(* IEC 61131-3 sources: Industry-PLC-LLM/data/PLCBEAD_repo/PLCBEAD_PLCEmbed-main/PLC-BEAD/Source/GEB/sample_project/oscat/Network, 47 files *)

(* ---- YAHOO_WEATHER_DESC_GE.ST ---- *)
TYPE
  oscat_STRING1               : STRING;
  oscat_STRING2               : STRING;
  oscat_STRING3               : STRING;
  oscat_STRING4               : STRING;
  oscat_STRING5               : STRING;
  oscat_STRING8               : STRING;
  oscat_STRING10              : STRING;
  oscat_STRING12            : STRING;
  oscat_STRING15            : STRING;
  oscat_STRING20            : STRING;
  oscat_STRING27            : STRING;
  oscat_STRING30            : STRING;
  oscat_STRING32            : STRING;
  oscat_STRING40            : STRING;
  oscat_STRING48            : STRING;
  oscat_STRING50            : STRING;
  oscat_STRING60            : STRING;
  oscat_STRING64            : STRING;
  oscat_STRING80            : STRING;
  oscat_STRING120            : STRING;
  oscat_STRING140            : STRING;
  oscat_STRING160            : STRING;
  oscat_STRING180            : STRING;
  oscat_STRING190            : STRING;
  oscat_STRING250            : STRING;
END_TYPE

TYPE
  oscat_IP_FIFO128_DATA  : ARRAY [1..128] OF BYTE;
  oscat_Mailbox  : ARRAY [1..16] OF BYTE;

  oscat_IP_FIFO_DATA :
  STRUCT
	X       : oscat_IP_FIFO128_DATA; (* IP_ID FIFO Speicher          *)
	Y       : oscat_IP_FIFO128_DATA; (* IP_ID Z�hler                 *)
	ID      : BYTE;                  (* h�chste vergabene id         *)
	MAX_ID  : BYTE;                  (* maximal Anmeldungen pro ID   *)
    INIT    : BOOL;                  (* Initialisierung durchgef�hrt *)
	EMPTY   : BOOL;                  (* FIFO leer                    *)
	FULL    : BOOL;                  (* FIFO voll                    *)
	TOP     : INT;                   (* maximale anzahl IN FIFO      *)
	NW      : INT;                   (* Schreibzeiger                *)
	NR      : INT;                   (* Lesezeiger                   *)
  END_STRUCT;

  oscat_IP_C:
  STRUCT
  	C_MODE:			BYTE;          		(*W Mode: TCP/UCP AKTIV/PASSIV                               *)
	C_PORT:         WORD;          		(*W Portnummer                                               *)
	C_IP:           DWORD;         		(*W IP-ADRESSe gepackt wwxxyyzz = www.xxx.yyy.zzz            *)
    C_STATE:        BYTE;          		(*R VerbindungsSTATUS ON/OFF + Flanke ON/OFF                 *)
	C_ENABLE:       BOOL;          		(*W Freigabe f�r Connect                                     *)
    R_OBSERVE:      BOOL;          		(*W Empfang ueberwachen                                      *)
    TIME_RESET:     BOOL;          		(*W Alle Timer ruecksetzen                                   *)
	ERROR:          DWORD;         		(*R vvwwxxyy (vv = CON_ERROR, ww = SEN_ERROR, xx = REC_ERROR *)
    FIFO:           oscat_IP_FIFO_DATA; (*I IP FIFO Struktur                                         *)
	MAILBOX:		oscat_Mailbox;		(*I Mailbox: Datenbereich f�r Bausteindatenaustausch         *)
  END_STRUCT;

  oscat_XML_CONTROL:
  STRUCT
    COMMAND:             WORD;            (*W                 *)
    WATCHDOG:            TIME;            (*W                 *)
    START_POS:           UINT;            (*W                 *)
    STOP_POS:            UINT;            (*W                 *)
    COUNT:               UINT;            (*R                 *)
    TYP:                 INT;             (*R                 *)
    LEVEL:               UINT;            (*R                 *)
    PATH:                oscat_STRING250; (*R                 *)
    ELEMENT:             oscat_STRING250; (*R                 *)
    ATTRIBUTE:           oscat_STRING250; (*R                 *)
    VALUE:               oscat_STRING250; (*R                 *)
    BLOCK1_START:        UINT;            (*R                 *)
    BLOCK1_STOP:         UINT;            (*R                 *)
    BLOCK2_START:        UINT;            (*R                 *)
    BLOCK2_STOP:         UINT;            (*R                 *)
  END_STRUCT;

  (* --------- WORLD WEATHER --------- *)

  oscat_WORLD_WEATHER_CUR :
  STRUCT
	OBSERVATION_TIME : oscat_STRING8;
	TEMP_C           : INT;
	WEATHER_CODE     : INT;
	WEATHER_DESC 	 : oscat_STRING60;
	WEATHER_ICON     : INT;
	WIND_SPEED_MILES : INT;
	WIND_SPEED_KMPH  : INT;
	WIND_DIR_DEGREE  : INT;
	WIND_DIR1 6POINT  : oscat_STRING3;
	PRECIPMM         : REAL;
	HUMIDITY         : INT;
	VISIBILITY       : INT;
	PRESSURE         : INT;
	CLOUDOVER        : INT;
  END_STRUCT;

  oscat_WORLD_WEATHER_DAY  :
  STRUCT
	DATE_OF_DAY       : oscat_STRING10;
	TEMP_MAX_C       : INT;
	TEMP_MAX_F       : INT;
	TEMP_MIN_C       : INT;
	TEMP_MIN_F       : INT;
	WIND_SPEED_MILES : INT;
	WIND_SPEED_KMPH  : INT;
	WIND_DIR_DEGREE  : INT;
	WIND_DIR1 6POINT  : oscat_STRING3;
	WEATHER_CODE     : INT;
	WEATHER_DESC     : oscat_STRING60;
	WEATHER_ICON     : INT;
	PRECIPMM         : REAL;
  END_STRUCT;

  oscat_WORLD_WEATHER_DAY_ARR : ARRAY [0..4] OF oscat_WORLD_WEATHER_DAY;

  oscat_WORLD_WEATHER_DATA :
  STRUCT
	CUR : oscat_WORLD_WEATHER_CUR;
	DAY  : oscat_WORLD_WEATHER_DAY_ARR;
  END_STRUCT;

  oscat_WORLD_WEATHER_aI0_41 : ARRAY[0..41] OF INT;

  (* --------- WEATHER CHANNEL --------- *)
  oscat_YAHOO_WEATHER_DATA:
  STRUCT
    TIMETOLIVE:                 INT;              (* TIME TO LIVE: HOW LONG IN MINUTES THIS FEED SHOULD BE CACHED         *)
    LOCATION_CITY:              OSCAT_STRING40;   (* THE LOCATION OF THIS FORECAST: CITY: CITY NAME  *)
    LOCATION_REGION:            OSCAT_STRING20;   (* THE LOCATION OF THIS FORECAST: REGION: STATE, TERRITORY, OR REGION, IF GIVEN *)
    LOCATION_COUNTRY:           OSCAT_STRING20;    (* THE LOCATION OF THIS FORECAST: COUNTRY: TWO-CHARACTER COUNTRY CODE *)
    UNIT_TEMPERATURE:           OSCAT_STRING1;    (* TEMPERATURE: DEGREE UNITS, F FOR FAHRENHEIT OR C FOR CELSIUS *)
    UNIT_DISTANCE:              OSCAT_STRING2;    (* DISTANCE: UNITS FOR DISTANCE, MI FOR MILES OR KM FOR KILOMETERS *)
    UNIT_PRESSURE:              OSCAT_STRING2;    (* PRESSURE: UNITS OF BAROMETRIC PRESSURE, IN FOR POUNDS PER SQUARE INCH OR MB FOR MILLIBARS *)
    UNIT_SPEED:                 OSCAT_STRING4;    (* SPEED: UNITS OF SPEED, MPH FOR MILES PER HOUR OR KPH FOR KILOMETERS PER HOUR *)
    WIND_CHILL:                 INT;              (* FORECAST INFORMATION ABOUT WIND CHILL IN DEGREES *)
    WIND_DIRECTION:             INT;              (* FORECAST INFORMATION ABOUT WIND DIRECTION, IN DEGREES *)
    WIND_SPEED:                 REAL;             (* FORECAST INFORMATION ABOUT WIND SPEED, IN THE UNITS (MPH OR KPH)*)
    ATMOSPHERE_HUMIDITY:        INT;              (* FORECAST INFORMATION ABOUT CURRENT ATMOSPHERIC HUMIDITY: HUMIDITY, IN PERCENT  *)
    ATMOSPHERE_PRESSURE:        INT;              (* FORECAST INFORMATION ABOUT CURRENT ATMOSPHERIC PRESSURE: BAROMETRIC PRESSURE, IN THE UNITS (IN OR MB) *)
	ATMOSPHERE_VISIBILITY:      REAL;             (* FORECAST INFORMATION ABOUT CURRENT ATMOSPHERIC VISIBILITY, IN THE UNITS (MI OR KM) *)
	ATMOSPHERE_RISING:          INT;              (* FORECAST INFORMATION ABOUT RISING: STATE OF THE BAROMETRIC PRESSURE: STEADY (0), RISING (1), OR FALLING (2). (INTEGER: 0, 1, 2) *)
    ASTRONOMY_SUNRISE:          OSCAT_STRING10;   (* SUNRISE: ToDAY'S SUNRISE TIME. THE TIME IS A STRING IN A LOCAL TIME FORMAT OF "H:MM AM/PM" *)
    ASTRONOMY_SUNSET:           OSCAT_STRING10;   (* SUNSET: ToDAY'S SUNSET TIME. THE TIME IS A STRING IN A LOCAL TIME FORMAT OF "H:MM AM/PM", *)
    GEO_LATITUDE:               REAL;             (* THE LATITUDE OF THE LOCATION *)
    GEO_LONGITUDE:              REAL;             (* THE LONGITUDE OF THE LOCATION *)
    CUR_CONDITIONS_TEMP:        INT;              (* THE CURRENT WEATHER CONDITIONS: TEMP: THE CURRENT TEMPERATURE, IN THE UNITS (F OR C) *)
    CUR_CONDITIONS_TEXT:        OSCAT_STRING40;   (* THE CURRENT WEATHER CONDITIONS: TEXT: A TEXTUAL DESCRIPTION OF CONDITIONS *)
    CUR_CONDITIONS_CODE:        INT;              (* THE CURRENT WEATHER CONDITIONS: CODE: THE CONDITION CODE FOR THIS FORECAST *)
	CUR_CONDITIONS_ICON:        INT;			  (* THE CURRENT WEATHER CONDITIONS: ICON: THE CONDITION ICON FOR THIS FORECAST *)
    FORCAST_ToDAY_LOW_TEMP:     INT;              (* THE FORCAST ToDAY  WEATHER CONDITIONS: THE FORECASTED LOW TEMPERATURE FOR THIS DAY  IN THE UNITS (F OR C) *)
    FORCAST_ToDAY_HIGH_TEMP:    INT;              (* THE FORCAST ToDAY  WEATHER CONDITIONS: THE FORECASTED HIGH TEMPERATURE FOR THIS DAY  IN THE UNITS (F OR C) *)
    FORCAST_ToDAY_TEXT:         OSCAT_STRING40;   (* THE FORCAST ToDAY  WEATHER CONDITIONS: TEXT: A TEXTUAL DESCRIPTION OF CONDITIONS *)
    FORCAST_ToDAY_CODE:         INT;              (* THE CURRENT WEATHER CONDITIONS: CODE: THE CONDITION CODE FOR THIS FORECAST *)
	FORCAST_ToDAY_ICON:         INT;			  (* THE CURRENT WEATHER CONDITIONS: ICON: THE CONDITION ICON FOR THIS FORECAST *)
    FORCAST_TOMORROW_LOW_TEMP:  INT;              (* THE FORCAST TOMORROW WEATHER CONDITIONS: THE FORECASTED LOW TEMPERATURE FOR THIS DAY  IN THE UNITS (F OR C) *)
    FORCAST_TOMORROW_HIGH_TEMP: INT;              (* THE FORCAST TOMORROW WEATHER CONDITIONS: THE FORECASTED HIGH TEMPERATURE FOR THIS DAY  IN THE UNITS (F OR C) *)
    FORCAST_TOMORROW_TEXT:      OSCAT_STRING40;   (* THE FORCAST TOMORROW WEATHER CONDITIONS: TEXT: A TEXTUAL DESCRIPTION OF CONDITIONS *)
    FORCAST_TOMORROW_CODE:      INT;              (* THE CURRENT WEATHER CONDITIONS: CODE: THE CONDITION CODE FOR THIS FORECAST *)
	FORCAST_TOMORROW_ICON:      INT;			  (* THE CURRENT WEATHER CONDITIONS: ICON: THE CONDITION ICON FOR THIS FORECAST *)
  END_STRUCT;

  oscat_YAHOO_WEATHER_aI0_48 : ARRAY[0..48] OF INT;

  oscat_IP2GEO_DATA:
  STRUCT
	STATE :				BOOL;			  (* STATE *)
	IP4 :				DWORD;			  (* IP-ADRESSe *)
    COUNTRY_CODE :		oscat_STRING2;    (*   *)
    COUNTRY_NAME :		oscat_STRING20;   (*   *)
    REGION_CODE :		oscat_STRING2;    (*   *)
    REGION_NAME :		oscat_STRING20;   (*   *)
    CITY :				oscat_STRING20;   (*   *)
    GEO_LATITUDE :		REAL;             (*   *)
    GEO_LONGITUDE :		REAL;             (*   *)
	TIME_ZONE_NAME :	oscat_STRING20;
	GMT_OFFSET :		INT;
	IS_DST :			BOOL;
  END_STRUCT;
END_TYPE

FUNCTION_BLOCK YAHOO_WEATHER_DESC_GE_Block

	VAR_INPUT
		ACTIVATE :	BOOL;
	END_VAR

	VAR_IN_OUT
		YW :	oscat_YAHOO_WEATHER_DATA;
	END_VAR

	VAR
		aCT_LAST :	BOOL;
		x :	INT;
		y :	INT;
		str :	oscat_STRING40;
	END_VAR

	IF ACTIVATE AND aCT_LAST = FALSE THEN
		FOR y := 1 TO 4 DO
			CASE y OF
			1:	x := YW.CUR_CONDITIONS_CODE;
			2 :	YW.CUR_CONDITIONS_TEXT := str;
				x := YW.FORCAST_ToDAY_CODE;
			3 :	YW.FORCAST_ToDAY_TEXT := str;
				x := YW.FORCAST_TOMORROW_CODE;
			4 :	YW.FORCAST_TOMORROW_TEXT := str;
			END_CASE;

			CASE x OF
			00:	str := 'Wirbelsturm';
			01:	str := 'Tropensturm';
			02:	str := 'Wirbelsturm';
			03:	str := 'starkes Gewitter ';
			04:	str := 'Gewitter';
			05:	str := 'Schneeregen';
			06:	str := 'Schneeregen';
			07:	str := 'Schneeregen';
			08:	str := 'gefrierender Nieselregen';
			09:	str := 'Nieselregen';
			10:	str := 'gefrierender Regen';
			11:	str := 'sertsehn';
			12:	str := 'sertstrets';
			13:	str := 'sjstj';
			14:	str := 'leichte yrderew';
			15:	str := 'Schneetreiben';
			16:	str := 'Schnee';
			17:	str := 'Hagel';
			18:	str := 'Schneeregen';
			19:	str := 'Staub';
			20:	str := 'nebelig';
			21:	str := 'Dunst';
			22:	str := 'rauchig';
			23:	str := 'sertsert';
			24:	str := 'windig';
			25:	str := 'kalt';
			26:	str := 'sertsert';
			27:	str := 'meist sertsert';
			28:	str := 'meist sertsert';
			29:	str := 'teilweise serhser';
			30:	str := 'teilweise sertsertshe';
			31:	str := 'klar';
			32:	str := 'sonnig';
			33:	str := 'heiter';
			34:	str := 'heiter';
			35:	str := 'Regen und Hagel';
			36:	str := 'WRYTWRYH';
			37:	str := 'esrertsertr';
			38:	str := 'vereinzelte Gewitter';
			39:	str := 'vereinzelte Gewitter';
			40:	str := 'verteesr';
			41:	str := 'sjstjtj';
			42:	str := 'sertsert';
			43:	str := 'sertsert';
			44:	str := 'sertsert';
			45:	str := 'sertsert';
			46:	str := 'sertsert';
			47:	str := 'srtsert';
			ELSE
				str := 'sertsert';
			END_CASE;
		END_FOR;
	END_IF;
	aCT_LAST := ACTIVATE;

END_FUNCTION_BLOCK

PROGRAM program0
	VAR
		ACTIVATE :	BOOL;
		YW :	oscat_YAHOO_WEATHER_DATA;

		func_block : YAHOO_WEATHER_DESC_GE_Block;
	END_VAR
	func_block.ACTIVATE := ACTIVATE;
	func_block.YW := YW;

	func_block();
	YW  := func_block.YW;
END_PROGRAM

CONFIGURATION Config0
	RESOURCE ReS0 ON PLC
		TASK task0(INTERVAL := T#20ms,PRIORITY := 0);
		PROGRAM instance0 WITH task0 : program0;
	END_RESOURCE
END_CONFIGURATION

(* ---- YAHOO_WEATHER_ICON_OSCAT.ST ---- *)
TYPE
  oscat_STRING1               : STRING;
  oscat_STRING2               : STRING;
  oscat_STRING3               : STRING;
  oscat_STRING4               : STRING;
  oscat_STRING5               : STRING;
  oscat_STRING8               : STRING;
  oscat_STRING10              : STRING;
  oscat_STRING12            : STRING;
  oscat_STRING15            : STRING;
  oscat_STRING20            : STRING;
  oscat_STRING27            : STRING;
  oscat_STRING30            : STRING;
  oscat_STRING32            : STRING;
  oscat_STRING40            : STRING;
  oscat_STRING48            : STRING;
  oscat_STRING50            : STRING;
  oscat_STRING60            : STRING;
  oscat_STRING64            : STRING;
  oscat_STRING80            : STRING;
  oscat_STRING120            : STRING;
  oscat_STRING140            : STRING;
  oscat_STRING160            : STRING;
  oscat_STRING180            : STRING;
  oscat_STRING190            : STRING;
  oscat_STRING250            : STRING;
END_TYPE

TYPE
  oscat_IP_FIFO128_DATA  : ARRAY [1..128] OF BYTE;
  oscat_Mailbox  : ARRAY [1..16] OF BYTE;

  oscat_IP_FIFO_DATA :
  STRUCT
	X       : oscat_IP_FIFO128_DATA; (* IP_ID FIFO Speicher          *)
	Y       : oscat_IP_FIFO128_DATA; (* IP_ID Z�hler                 *)
	ID      : BYTE;                  (* h�chste vergabene id         *)
	MAX_ID  : BYTE;                  (* maximal Anmeldungen pro ID   *)
    INIT    : BOOL;                  (* Initialisierung durchgef�hrt *)
	EMPTY   : BOOL;                  (* FIFO leer                    *)
	FULL    : BOOL;                  (* FIFO voll                    *)
	TOP     : INT;                   (* maximale anzahl IN FIFO      *)
	NW      : INT;                   (* Schreibzeiger                *)
	NR      : INT;                   (* Lesezeiger                   *)
  END_STRUCT;

  oscat_IP_C:
  STRUCT
  	C_MODE:			BYTE;          		(*W Mode: TCP/UCP AKTIV/PASSIV                               *)
	C_PORT:         WORD;          		(*W Portnummer                                               *)
	C_IP:           DWORD;         		(*W IP-ADRESSe gepackt wwxxyyzz = www.xxx.yyy.zzz            *)
    C_STATE:        BYTE;          		(*R VerbindungsSTATUS ON/OFF + Flanke ON/OFF                 *)
	C_ENABLE:       BOOL;          		(*W Freigabe f�r Connect                                     *)
    R_OBSERVE:      BOOL;          		(*W Empfang ueberwachen                                      *)
    TIME_RESET:     BOOL;          		(*W Alle Timer ruecksetzen                                   *)
	ERROR:          DWORD;         		(*R vvwwxxyy (vv = CON_ERROR, ww = SEN_ERROR, xx = REC_ERROR *)
    FIFO:           oscat_IP_FIFO_DATA; (*I IP FIFO Struktur                                         *)
	MAILBOX:		oscat_Mailbox;		(*I Mailbox: Datenbereich f�r Bausteindatenaustausch         *)
  END_STRUCT;

  oscat_XML_CONTROL:
  STRUCT
    COMMAND:             WORD;            (*W                 *)
    WATCHDOG:            TIME;            (*W                 *)
    START_POS:           UINT;            (*W                 *)
    STOP_POS:            UINT;            (*W                 *)
    COUNT:               UINT;            (*R                 *)
    TYP:                 INT;             (*R                 *)
    LEVEL:               UINT;            (*R                 *)
    PATH:                oscat_STRING250; (*R                 *)
    ELEMENT:             oscat_STRING250; (*R                 *)
    ATTRIBUTE:           oscat_STRING250; (*R                 *)
    VALUE:               oscat_STRING250; (*R                 *)
    BLOCK1_START:        UINT;            (*R                 *)
    BLOCK1_STOP:         UINT;            (*R                 *)
    BLOCK2_START:        UINT;            (*R                 *)
    BLOCK2_STOP:         UINT;            (*R                 *)
  END_STRUCT;

  (* --------- WORLD WEATHER --------- *)

  oscat_WORLD_WEATHER_CUR :
  STRUCT
	OBSERVATION_TIME : oscat_STRING8;
	TEMP_C           : INT;
	WEATHER_CODE     : INT;
	WEATHER_DESC 	 : oscat_STRING60;
	WEATHER_ICON     : INT;
	WIND_SPEED_MILES : INT;
	WIND_SPEED_KMPH  : INT;
	WIND_DIR_DEGREE  : INT;
	WIND_DIR1 6POINT  : oscat_STRING3;
	PRECIPMM         : REAL;
	HUMIDITY         : INT;
	VISIBILITY       : INT;
	PRESSURE         : INT;
	CLOUDOVER        : INT;
  END_STRUCT;

  oscat_WORLD_WEATHER_DAY  :
  STRUCT
	DATE_OF_DAY       : oscat_STRING10;
	TEMP_MAX_C       : INT;
	TEMP_MAX_F       : INT;
	TEMP_MIN_C       : INT;
	TEMP_MIN_F       : INT;
	WIND_SPEED_MILES : INT;
	WIND_SPEED_KMPH  : INT;
	WIND_DIR_DEGREE  : INT;
	WIND_DIR1 6POINT  : oscat_STRING3;
	WEATHER_CODE     : INT;
	WEATHER_DESC     : oscat_STRING60;
	WEATHER_ICON     : INT;
	PRECIPMM         : REAL;
  END_STRUCT;

  oscat_WORLD_WEATHER_DAY_ARR : ARRAY [0..4] OF oscat_WORLD_WEATHER_DAY;

  oscat_WORLD_WEATHER_DATA :
  STRUCT
	CUR : oscat_WORLD_WEATHER_CUR;
	DAY  : oscat_WORLD_WEATHER_DAY_ARR;
  END_STRUCT;

  oscat_WORLD_WEATHER_aI0_41 : ARRAY[0..41] OF INT;

  (* --------- WEATHER CHANNEL --------- *)
  oscat_YAHOO_WEATHER_DATA:
  STRUCT
    TIMETOLIVE:                 INT;              (* TIME TO LIVE: HOW LONG IN MINUTES THIS FEED SHOULD BE CACHED         *)
    LOCATION_CITY:              OSCAT_STRING40;   (* THE LOCATION OF THIS FORECAST: CITY: CITY NAME  *)
    LOCATION_REGION:            OSCAT_STRING20;   (* THE LOCATION OF THIS FORECAST: REGION: STATE, TERRITORY, OR REGION, IF GIVEN *)
    LOCATION_COUNTRY:           OSCAT_STRING20;    (* THE LOCATION OF THIS FORECAST: COUNTRY: TWO-CHARACTER COUNTRY CODE *)
    UNIT_TEMPERATURE:           OSCAT_STRING1;    (* TEMPERATURE: DEGREE UNITS, F FOR FAHRENHEIT OR C FOR CELSIUS *)
    UNIT_DISTANCE:              OSCAT_STRING2;    (* DISTANCE: UNITS FOR DISTANCE, MI FOR MILES OR KM FOR KILOMETERS *)
    UNIT_PRESSURE:              OSCAT_STRING2;    (* PRESSURE: UNITS OF BAROMETRIC PRESSURE, IN FOR POUNDS PER SQUARE INCH OR MB FOR MILLIBARS *)
    UNIT_SPEED:                 OSCAT_STRING4;    (* SPEED: UNITS OF SPEED, MPH FOR MILES PER HOUR OR KPH FOR KILOMETERS PER HOUR *)
    WIND_CHILL:                 INT;              (* FORECAST INFORMATION ABOUT WIND CHILL IN DEGREES *)
    WIND_DIRECTION:             INT;              (* FORECAST INFORMATION ABOUT WIND DIRECTION, IN DEGREES *)
    WIND_SPEED:                 REAL;             (* FORECAST INFORMATION ABOUT WIND SPEED, IN THE UNITS (MPH OR KPH)*)
    ATMOSPHERE_HUMIDITY:        INT;              (* FORECAST INFORMATION ABOUT CURRENT ATMOSPHERIC HUMIDITY: HUMIDITY, IN PERCENT  *)
    ATMOSPHERE_PRESSURE:        INT;              (* FORECAST INFORMATION ABOUT CURRENT ATMOSPHERIC PRESSURE: BAROMETRIC PRESSURE, IN THE UNITS (IN OR MB) *)
	ATMOSPHERE_VISIBILITY:      REAL;             (* FORECAST INFORMATION ABOUT CURRENT ATMOSPHERIC VISIBILITY, IN THE UNITS (MI OR KM) *)
	ATMOSPHERE_RISING:          INT;              (* FORECAST INFORMATION ABOUT RISING: STATE OF THE BAROMETRIC PRESSURE: STEADY (0), RISING (1), OR FALLING (2). (INTEGER: 0, 1, 2) *)
    ASTRONOMY_SUNRISE:          OSCAT_STRING10;   (* SUNRISE: ToDAY'S SUNRISE TIME. THE TIME IS A STRING IN A LOCAL TIME FORMAT OF "H:MM AM/PM" *)
    ASTRONOMY_SUNSET:           OSCAT_STRING10;   (* SUNSET: ToDAY'S SUNSET TIME. THE TIME IS A STRING IN A LOCAL TIME FORMAT OF "H:MM AM/PM", *)
    GEO_LATITUDE:               REAL;             (* THE LATITUDE OF THE LOCATION *)
    GEO_LONGITUDE:              REAL;             (* THE LONGITUDE OF THE LOCATION *)
    CUR_CONDITIONS_TEMP:        INT;              (* THE CURRENT WEATHER CONDITIONS: TEMP: THE CURRENT TEMPERATURE, IN THE UNITS (F OR C) *)
    CUR_CONDITIONS_TEXT:        OSCAT_STRING40;   (* THE CURRENT WEATHER CONDITIONS: TEXT: A TEXTUAL DESCRIPTION OF CONDITIONS *)
    CUR_CONDITIONS_CODE:        INT;              (* THE CURRENT WEATHER CONDITIONS: CODE: THE CONDITION CODE FOR THIS FORECAST *)
	CUR_CONDITIONS_ICON:        INT;			  (* THE CURRENT WEATHER CONDITIONS: ICON: THE CONDITION ICON FOR THIS FORECAST *)
    FORCAST_ToDAY_LOW_TEMP:     INT;              (* THE FORCAST ToDAY  WEATHER CONDITIONS: THE FORECASTED LOW TEMPERATURE FOR THIS DAY  IN THE UNITS (F OR C) *)
    FORCAST_ToDAY_HIGH_TEMP:    INT;              (* THE FORCAST ToDAY  WEATHER CONDITIONS: THE FORECASTED HIGH TEMPERATURE FOR THIS DAY  IN THE UNITS (F OR C) *)
    FORCAST_ToDAY_TEXT:         OSCAT_STRING40;   (* THE FORCAST ToDAY  WEATHER CONDITIONS: TEXT: A TEXTUAL DESCRIPTION OF CONDITIONS *)
    FORCAST_ToDAY_CODE:         INT;              (* THE CURRENT WEATHER CONDITIONS: CODE: THE CONDITION CODE FOR THIS FORECAST *)
	FORCAST_ToDAY_ICON:         INT;			  (* THE CURRENT WEATHER CONDITIONS: ICON: THE CONDITION ICON FOR THIS FORECAST *)
    FORCAST_TOMORROW_LOW_TEMP:  INT;              (* THE FORCAST TOMORROW WEATHER CONDITIONS: THE FORECASTED LOW TEMPERATURE FOR THIS DAY  IN THE UNITS (F OR C) *)
    FORCAST_TOMORROW_HIGH_TEMP: INT;              (* THE FORCAST TOMORROW WEATHER CONDITIONS: THE FORECASTED HIGH TEMPERATURE FOR THIS DAY  IN THE UNITS (F OR C) *)
    FORCAST_TOMORROW_TEXT:      OSCAT_STRING40;   (* THE FORCAST TOMORROW WEATHER CONDITIONS: TEXT: A TEXTUAL DESCRIPTION OF CONDITIONS *)
    FORCAST_TOMORROW_CODE:      INT;              (* THE CURRENT WEATHER CONDITIONS: CODE: THE CONDITION CODE FOR THIS FORECAST *)
	FORCAST_TOMORROW_ICON:      INT;			  (* THE CURRENT WEATHER CONDITIONS: ICON: THE CONDITION ICON FOR THIS FORECAST *)
  END_STRUCT;

  oscat_YAHOO_WEATHER_aI0_48 : ARRAY[0..48] OF INT;

  oscat_IP2GEO_DATA:
  STRUCT
	STATE :				BOOL;			  (* STATE *)
	IP4 :				DWORD;			  (* IP-ADRESSe *)
    COUNTRY_CODE :		oscat_STRING2;    (*   *)
    COUNTRY_NAME :		oscat_STRING20;   (*   *)
    REGION_CODE :		oscat_STRING2;    (*   *)
    REGION_NAME :		oscat_STRING20;   (*   *)
    CITY :				oscat_STRING20;   (*   *)
    GEO_LATITUDE :		REAL;             (*   *)
    GEO_LONGITUDE :		REAL;             (*   *)
	TIME_ZONE_NAME :	oscat_STRING20;
	GMT_OFFSET :		INT;
	IS_DST :			BOOL;
  END_STRUCT;
END_TYPE

FUNCTION_BLOCK YAHOO_WEATHER_ICON_OSCAT_Block

	VAR_INPUT
		ACTIVATE :	BOOL;
	END_VAR

	VAR_IN_OUT
		YW :	oscat_YAHOO_WEATHER_DATA;
	END_VAR

	VAR
		aCT_LAST :	BOOL;
		x :	INT;
		init :	BOOL;
		dat :	oscat_YAHOO_WEATHER_aI0_48;
	END_VAR

	IF not init THEN
		init := TRUE;

		dat[00] := 4;
		dat[01] := 2;
		dat[02] := 2;
		dat[03] := 4;
		dat[04] := 17;
		dat[05] := 1;
		dat[06] := 3;
		dat[07] := 1;
		dat[08] := 2;
		dat[09] := 2;
		dat[10] := 2;
		dat[11] := 2;
		dat[12] := 2;
		dat[13] := 3;
		dat[14] := 3;
		dat[15] := 3;
		dat[16] := 3;
		dat[17] := 5;
		dat[18] := 3;
		dat[19] := 6;
		dat[20] := 7;
		dat[21] := 14;
		dat[22] := 8;
		dat[23] := 9;
		dat[24] := 9;
		dat[25] := 10;
		dat[26] := 9;
		dat[27] := 11;
		dat[28] := 12;
		dat[29] := 11;
		dat[30] := 12;
		dat[31] := 13;
		dat[32] := 14;
		dat[33] := 15;
		dat[34] := 16;
		dat[35] := 4;
		dat[36] := 14;
		dat[37] := 4;
		dat[38] := 17;
		dat[39] := 2;
		dat[40] := 2;
		dat[41] := 3;
		dat[42] := 3;
		dat[43] := 3;
		dat[44] := 12;
		dat[45] := 2;
		dat[46] := 3;
		dat[47] := 4;
		dat[48] := 0;
	END_IF;

	IF ACTIVATE AND aCT_LAST = FALSE THEN
		x := MIN(YW.CUR_CONDITIONS_CODE,48);
		YW.CUR_CONDITIONS_ICON := dat[x];
		x := MIN(YW.FORCAST_ToDAY_CODE,48);
		YW.FORCAST_ToDAY_ICON := dat[x];
		x := MIN(YW.FORCAST_TOMORROW_CODE,48);
		YW.FORCAST_TOMORROW_ICON := dat[x];
	END_IF;
	aCT_LAST := ACTIVATE;

END_FUNCTION_BLOCK

PROGRAM program0
	VAR
		ACTIVATE :	BOOL;
		YW :	oscat_YAHOO_WEATHER_DATA;

		func_block : YAHOO_WEATHER_ICON_OSCAT_Block;
	END_VAR
	func_block.ACTIVATE := ACTIVATE;
	func_block.YW := YW;

	func_block();
	YW  := func_block.YW;
END_PROGRAM

CONFIGURATION Config0
	RESOURCE ReS0 ON PLC
		TASK task0(INTERVAL := T#20ms,PRIORITY := 0);
		PROGRAM instance0 WITH task0 : program0;
	END_RESOURCE
END_CONFIGURATION

(* ---- _BUFFER_UPPERCASE_NW.ST ---- *)
TYPE
  oscat_NW_BUF_LONG  : ARRAY [0..4095] OF BYTE;
END_TYPE

FUNCTION SETUP_EXTENDED_ASCII:BOOL
	VAR_INPUT
		X :	BOOL;
	END_VAR

	SETUP_EXTENDED_ASCII := X OR TRUE;
END_FUNCTION

FUNCTION TO_UPPER:BYTE

	VAR_INPUT
		IN :	BYTE;
	END_VAR

	IF IN > BYTE#96 AND IN < BYTE#123 THEN
	TO_UPPER := IN AND BYTE#16#DF;
	ELSIF IN > BYTE#223 AND IN <> BYTE#247 AND IN <> BYTE#255 AND SETUP_EXTENDED_ASCII(FALSE) THEN
	TO_UPPER := IN AND BYTE#16#DF;
	ELSE
	TO_UPPER := IN;
	END_IF;

END_FUNCTION

FUNCTION_BLOCK _BUFFER_UPPERCASE_NW
	VAR_INPUT
		SIZE :	UINT;
	END_VAR

	VAR_OUTPUT
		_BUFFER_UPPERCASE :	BOOL;
	END_VAR

	VAR_IN_OUT
		PT :	oscat_NW_BUF_LONG;
	END_VAR

	VAR
		POS :	INT;
		SIZE2 :	INT;
	END_VAR

	POS := 0;
	SIZE2 := UINT_TO_INT(SIZE);

	WHILE POS < SIZE2 DO
		PT[POS] := TO_UPPER(PT[POS]);
		POS := POS + 1;
	END_WHILE;

	_BUFFER_UPPERCASE := TRUE;

END_FUNCTION_BLOCK

PROGRAM program0
  VAR
	SIZE :	UINT;

	_BUFFER_UPPERCASE :	BOOL;

	PT :	oscat_NW_BUF_LONG;

	func_block : _BUFFER_UPPERCASE_NW;
  END_VAR
	func_block.SIZE  :=SIZE ;
	func_block.PT  :=PT ;
	func_block();
	PT := func_block.PT;
	_BUFFER_UPPERCASE := func_block._BUFFER_UPPERCASE;
END_PROGRAM

CONFIGURATION Config0
  RESOURCE ReS0 ON PLC
    TASK task0(INTERVAL := T#20ms,PRIORITY := 0);
    PROGRAM instance0 WITH task0 : program0;
  END_RESOURCE
END_CONFIGURATION

(* ---- BASE64_DECODE_STREAM.ST ---- *)
TYPE
  oscat_aB0_47	: ARRAY [0..47]	OF BYTE;
  oscat_aB0_63	: ARRAY [0..63]	OF BYTE;
END_TYPE

FUNCTION_BLOCK BASE64_DECODE_STREAM
	VAR_IN_OUT
		BUF1 :	oscat_aB0_63;
		BUF2 :	oscat_aB0_47;
	END_VAR

	VAR_INPUT
		SIZE1 :	INT;
	END_VAR

	VAR_OUTPUT
		SIZE2 :	INT;
	END_VAR

	VAR
		a :	INT;
		b :	WORD;
		o :	INT;
		off :	INT;
		i1 :	INT;
		i2 :	INT;
		c :	INT;
	END_VAR

	IF SIZE1 <= 0 THEN SIZE2 := 0; RETURN; END_IF;
	c := SIZE1 - 1;
	i2 := 0;
	a := 0;
	b := WORD#0;
	FOR i1 := 0 TO c DO
		o := BYTE_TO_INT(BUF1[i1]);
		IF o = 61  (* = *) THEN EXIT;
		ELSIF o > 96 (* a-z *) THEN off := 71;
		ELSIF o > 64 (* A-Z *) THEN off := 65;
		ELSIF o > 47 (* 0-9 *) THEN off := -4;
		ELSIF o = 43 (* + *) THEN off := -19;
		ELSIF o = 47 (* / *) THEN off := -16;
		END_IF;
		b := SHL(b,6) OR INT_TO_WORD(o - off);
		a := a + 6;
		IF a >= 8 THEN
			a := a - 8;
			BUF2[i2] := WORD_TO_BYTE(SHR(b,a));
			i2 := i2 + 1;
			b := b AND NOT SHL(WORD#16#FFFF,a);
		END_IF;
	END_FOR;
	SIZE2 := i2;
END_FUNCTION_BLOCK

PROGRAM program0
  VAR
	BUF1  :	oscat_aB0_63;
	BUF2  :	oscat_aB0_47;

	SIZE1 :	INT;

	SIZE2 :	INT;
	func_block : BASE64_DECODE_STREAM;
  END_VAR
	func_block.BUF1 :=BUF1 ;
	func_block.BUF2 :=BUF2 ;
	func_block.SIZE1:=SIZE1;
	func_block();
	BUF1 := func_block.BUF1;
	BUF2 := func_block.BUF2;
	SIZE2 := func_block.SIZE2;
END_PROGRAM

CONFIGURATION Config0
  RESOURCE ReS0 ON PLC
    TASK task0(INTERVAL := T#20ms,PRIORITY := 0);
    PROGRAM instance0 WITH task0 : program0;
  END_RESOURCE
END_CONFIGURATION

(* ---- BUFFER_COMP_NW.ST ---- *)
TYPE
  oscat_NW_BUF_LONG  : ARRAY [0..4095] OF BYTE;
END_TYPE

FUNCTION_BLOCK BUFFER_COMP_NW
	VAR_IN_OUT
		PT1 :	oscat_NW_BUF_LONG;
	END_VAR

	VAR_INPUT
		SIZE1 :	INT;
	END_VAR

	VAR_IN_OUT
		PT2 :	oscat_NW_BUF_LONG;
	END_VAR

	VAR_INPUT
		SIZE2 :	INT;
		START :	INT;
	END_VAR

	VAR_OUTPUT
		BUFFER_COMP :	INT;
	END_VAR

	VAR
		i :	INT;
		j :	INT;
		end :	INT;
		j2 :	INT;
	END_VAR

	IF SIZE2 <= SIZE1 AND SIZE1 > 0 AND SIZE2 > 0 AND START >= 0 THEN
		end := SIZE1 - SIZE2;
		FOR i := START TO end DO
			IF PT1[i] = PT2[0] THEN
				(* first CHARacter matches, now compare rest of array *)
				j := 1;
				j2 := j + i;
				WHILE j < SIZE2 DO
					IF PT2[j] <> PT1[j2] THEN EXIT; END_IF;
					j := j + 1;
					j2 := j2 + 1;
				END_WHILE;
				(* when J > SIZE2 a match was found return the POSition i IN buffeR1  *)
				IF j = SIZE2 THEN
					BUFFER_COMP := i;
					RETURN;
				END_IF;
			END_IF;
		END_FOR;
	END_IF;
	BUFFER_COMP := -1;

END_FUNCTION_BLOCK

PROGRAM program0
  VAR
	PT1   :	oscat_NW_BUF_LONG;

	SIZE1 :	INT;

	PT2   : 	oscat_NW_BUF_LONG;

	SIZE2 :	INT;
	START :	INT;

	BUFFER_COMP :	INT;

	func_block : BUFFER_COMP_NW;
  END_VAR
	func_block.PT1  :=PT1  ;
	func_block.SIZE1:=SIZE1;
	func_block.PT2  :=PT2  ;
	func_block.SIZE2:=SIZE2;
	func_block.START:=START;
	func_block();
	BUFFER_COMP := func_block.BUFFER_COMP;
	PT1 := func_block.PT1;
	PT2 := func_block.PT2;

END_PROGRAM

CONFIGURATION Config0
  RESOURCE ReS0 ON PLC
    TASK task0(INTERVAL := T#20ms,PRIORITY := 0);
    PROGRAM instance0 WITH task0 : program0;
  END_RESOURCE
END_CONFIGURATION

(* ---- FILE_BLOCK.ST ---- *)
TYPE
  oscat_FILE_SERVER_DATA : STRUCT
	FILE_OPEN	: BOOL;
    FILENAME 	: STRING;
    MODE	 	: BYTE;
    OFFSET   	: UDINT;
    FILE_SIZE   : UDINT;
    AUTO_CLOSE	: TIME;
    ERROR	 	: BYTE;
  END_STRUCT;

  oscat_NW_BUF_LONG  : ARRAY [0..4095] OF BYTE;
  oscat_NETWORK_BUFFER :
  STRUCT
    SIZE   : UINT;
    BUFFER : oscat_NW_BUF_LONG;
  END_STRUCT;
END_TYPE

FUNCTION_BLOCK FILE_BLOCK

	VAR_IN_OUT
		MODE :	BYTE;
		FILENAME :	STRING;
		FSD :	oscat_FILE_SERVER_DATA;
		PT :	oscat_NETWORK_BUFFER;
	END_VAR

	VAR_INPUT
		POS :	UDINT;
	END_VAR

	VAR_OUTPUT
		ERROR :	BYTE;
		DATA :	BYTE;
	END_VAR

	VAR
		STEPP :	INT;
		i :	INT;
		data_START :	UDINT;
		data_STOP :	UDINT;
	END_VAR

	CASE STEPP OF
	0:	IF MODE > BYTE#0 THEN
			ERROR := BYTE#0;
			IF FSD.FILE_OPEN AND (FSD.FILE_SIZE = UDINT#0 OR POS >= FSD.FILE_SIZE) THEN
				ERROR := BYTE#255;
				MODE := BYTE#0;
			ELSIF POS < data_START OR POS > data_STOP OR NOT FSD.FILE_OPEN THEN
				FSD.FILENAME := FILENAME;
				FSD.MODE := BYTE#1;
				FSD.OFFSET := POS;
				PT.SIZE := UINT#65535;
				data_START := UDINT#0;
				data_STOP := UDINT#0;
				STEPP := 10;
			ELSE
				i := UDINT_TO_INT(POS - data_START);
				DATA := PT.BUFFER[i];
				MODE := BYTE#0;
			END_IF;
		END_IF;

	10:	IF FSD.MODE = BYTE#0 THEN
			IF FSD.ERROR > BYTE#0 THEN
				ERROR := FSD.ERROR;
				MODE := BYTE#0;
			ELSE
				data_START := POS;
				data_STOP := POS + UINT_TO_UDINT(PT.SIZE) - UDINT#1;
			END_IF;
			STEPP := 0;
		END_IF;
	END_CASE;
END_FUNCTION_BLOCK

PROGRAM program0
	VAR
		MODE :	BYTE;
		FILENAME :	STRING;
		FSD :	oscat_FILE_SERVER_DATA;
		PT :	oscat_NETWORK_BUFFER;
		POS :	UDINT;
		ERROR :	BYTE;
		DATA :	BYTE;

		func_block : FILE_BLOCK;
	END_VAR
	func_block.MODE    :=MODE    ;
	func_block.FILENAME:=FILENAME;
	func_block.FSD     :=FSD     ;
	func_block.PT      :=PT      ;
	func_block.POS     :=POS     ;
	func_block();
	MODE    := func_block.MODE    ;
	FILENAME:= func_block.FILENAME;
	FSD     := func_block.FSD     ;
	PT      := func_block.PT      ;
	ERROR   := func_block.ERROR;
	DATA    := func_block.DATA;

END_PROGRAM

(* ---- FILE_PATH_SPLIT.ST ---- *)
TYPE
  oscat_STRING250             : STRING;
  oscat_STRING1             : STRING;
  oscat_STRING80             : STRING;
  oscat_STRING3             : STRING;
  oscat_NW_BUF_LONG  : ARRAY [0..4095] OF BYTE;
  PRINTF_DATA_250  	:  ARRAY [1..11]  OF oscat_STRING250;
  PRINTF_DATA_80 	:  ARRAY [1..11]  OF oscat_STRING80;
  LOG_250       	:  ARRAY [0..400] OF oscat_STRING250;
  LOG_80    		:  ARRAY [0..400] OF oscat_STRING80;
  LOG_OPTION		:  ARRAY [0..400] OF DWORD;

  us_LOG_CONTROL :
  STRUCT
    NEW_MSG              : oscat_STRING250;    (*W neue Nachricht f�r den Datenbuffer   *)
	NEW_MSG_OPTION 		 : DWORD;
    LEVEL                : BYTE;
	SIZE                 : INT;                (*R Anzahl der Strings im LOG_DATA       *)
	RESET                : BOOL;               (*W Nachrichtenbuffer l�schen            *)
    PRINTF               : PRINTF_DATA_250;    (*W Array PRINTF Parameter               *)
    MSG                  : LOG_250;            (*I Array Message                        *)
    MSG_OPTION           : LOG_OPTION;     	   (*I Array Message OPTion                 *)
	UPDATE_COUNT         : UINT;               (*R Updatez�hler                         *)
    IDX                  : INT;                (*R aktueller Nachrichten-Index          *)
	RING_MODE            : BOOL;               (*I Buffer�berlauf erkannt               *)
  END_STRUCT;

  us_LOG_CONTROL_80 :
  STRUCT
    NEW_MSG              : oscat_STRING80;     (*W neue Nachricht f�r den Datenbuffer   *)
	NEW_MSG_OPTION 		 : DWORD;
    LEVEL                : BYTE;
	SIZE                 : INT;                (*R Anzahl der Strings im LOG_DATA       *)
	RESET                : BOOL;               (*W Nachrichtenbuffer l�schen            *)
    PRINTF               : PRINTF_DATA_80;     (*W Array PRINTF Parameter               *)
    MSG                  : LOG_80;             (*I Array Message                        *)
    MSG_OPTION           : LOG_OPTION;     	   (*I Array Message OPTion                 *)
	UPDATE_COUNT         : UINT;               (*R Updatez�hler                         *)
    IDX                  : INT;                (*R aktueller Nachrichten-Index          *)
	RING_MODE            : BOOL;               (*I Buffer�berlauf erkannt               *)
  END_STRUCT;

  LINE_ARRAY 			: ARRAY [1..40] OF INT;

  us_LOG_VIEWPORT :
    STRUCT
     LINE_ARRAY          : LINE_ARRAY;
     COUNT               : INT;                (* Anzahl der sichtbaren Nachtrichten   *)
	 UPDATE_COUNT        : UINT;               (* Updatez�hler                         *)
     MOVE_TO_X           : INT;                (* Steuerung der Nachrichtenanzeige     *)
     UPDATE              : BOOL;               (* Daten wurden ge�ndert -> neuzeichnen *)
  END_STRUCT;

  oscat_FILE_SERVER_DATA : STRUCT
	FILE_OPEN	: BOOL;
    FILENAME 	: STRING;
    MODE	 	: BYTE;
    OFFSET   	: UDINT;
    FILE_SIZE   : UDINT;
    AUTO_CLOSE	: TIME;
    ERROR	 	: BYTE;
  END_STRUCT;

  oscat_FILE_PATH_DATA : STRUCT
	DRIVE : oscat_string3;
	DIRECTORY : oscat_string250;
	FILENAME : STRING;
  END_STRUCT;

  oscat_UNI_CIRCULAR_BUFFER_DATA : STRUCT
	D_MODE : INT;
	D_HEAD : WORD;
	D_STRING : oscat_string250;
	D_REAL : REAL;
	D_DWORD : DWORD;
	BUF_SIZE : INT;
	BUF_COUNT : INT;
	BUF_USED : USINT;
	BUF : oscat_NW_BUF_LONG;
	_GetSTART : INT;
	_GetEnd : INT;
	_Last : INT;
	_FiRST : INT;
  END_STRUCT;

  oscat_DLOG_DATA : STRUCT
	STORE_TYPE : BYTE;
	ADD_HEADER : BOOL;
	ADD_DATA : BOOL;
	ADD_DATA_REQ : BOOL;
	CLOCK_TRIG : BOOL;
	ID_MAX : USINT;
	DTI : UDINT;
	UCB : oscat_UNI_CIRCULAR_BUFFER_DATA;
	NEW_FILE : STRING;
	NEW_FILE_RTRIG : BOOL;
  END_STRUCT;

END_TYPE

FUNCTION_BLOCK FILE_PATH_SPLIT_Block

	VAR_INPUT
		FILENAME :	oscat_STRING250;
	END_VAR

	VAR_OUTPUT
		FILE_PATH_SPLIT :	BOOL;
	END_VAR

	VAR_IN_OUT
		X :	oscat_FILE_PATH_DATA;
	END_VAR

	VAR
		b :	INT;
		c :	INT;
		d :	oscat_STRING1;
		p1 :	INT;
		p2 :	INT;
	END_VAR

	X.DRIVE := '';
	X.DIRECTORY := '';
	X.FILENAME := '';
	p1 := 0;
	p2 := 0;
	c := LEN(FILENAME);
	IF c = 0 THEN
		FILE_PATH_SPLIT := FALSE;
		RETURN;
	END_IF;

	FOR b := 1 TO c DO
		d := MID(FILENAME, 1, b);
		IF EQ_STRING(d,':') THEN
			p1 := b;
		ELSIF EQ_STRING(d,'/') OR EQ_STRING(d,'\') THEN
			p2 := b;
		END_IF;
	END_FOR;

	IF p1 = 2 THEN
		X.DRIVE := LEFT(FILENAME,p1);
	END_IF;

	IF p2 > 0 AND p2 > p1 THEN
		X.DIRECTORY := MID(FILENAME,p2-p1,p1+1);
	END_IF;

	X.FILENAME := RIGHT(FILENAME,c - MAX (p1,p2));
	FILE_PATH_SPLIT := TRUE;

END_FUNCTION_BLOCK

PROGRAM program0
	VAR
		FILENAME :	oscat_STRING250;
		FILE_PATH_SPLIT :	BOOL;
		X :	oscat_FILE_PATH_DATA;

		func_block : FILE_PATH_SPLIT_Block;
	END_VAR
	func_block.FILENAME := FILENAME;
	func_block.X := X;

	func_block();
	FILE_PATH_SPLIT  := func_block.FILE_PATH_SPLIT;
	X  := func_block.X;
END_PROGRAM

CONFIGURATION Config0
	RESOURCE ReS0 ON PLC
		TASK task0(INTERVAL := T#20ms,PRIORITY := 0);
		PROGRAM instance0 WITH task0 : program0;
	END_RESOURCE
END_CONFIGURATION

(* ---- IP4_TO_STRING.ST ---- *)
TYPE
  oscat_STRING10             : STRING;
END_TYPE

FUNCTION _BYTE_TO_INT:INT
	VAR_INPUT
		IN :	BYTE;
	END_VAR

	_BYTE_TO_INT := USINT_TO_INT(BYTE_TO_USINT(IN));
END_FUNCTION

FUNCTION BYTE_OF_DWORD:BYTE
	VAR_INPUT
		IN :	DWORD;
		N :	BYTE;
	END_VAR
	BYTE_OF_DWORD := DWORD_TO_BYTE(SHR(IN,_BYTE_TO_INT(SHL(n,3))));
END_FUNCTION

FUNCTION_BLOCK IP4_TO_STRING_Block

	VAR_INPUT
		IP4 :	DWORD;
	END_VAR

	VAR_OUTPUT
		IP4_TO_STRING :	STRING;
	END_VAR

	VAR
		S1 :	oscat_string10;
		S2 :	oscat_string10;
	END_VAR

	S1 := CONCAT(BYTE_TO_STRING(BYTE_OF_DWORD(IP4,BYTE#1)),BYTE_TO_STRING(BYTE_OF_DWORD(IP4,BYTE#0)));
	S2 := CONCAT(BYTE_TO_STRING(BYTE_OF_DWORD(IP4,BYTE#3)),BYTE_TO_STRING(BYTE_OF_DWORD(IP4,BYTE#2)));
	IP4_TO_STRING := CONCAT(S2,S1);

END_FUNCTION_BLOCK

PROGRAM program0
	VAR
		IP4 :	DWORD;
		IP4_TO_STRING :	STRING;

		func_block : IP4_TO_STRING_Block;
	END_VAR
	func_block.IP4 := IP4;

	func_block();
	IP4_TO_STRING  := func_block.IP4_TO_STRING;
END_PROGRAM

CONFIGURATION Config0

  	RESOURCE ReS0 ON PLC
    	TASK task0(INTERVAL := T#20ms,PRIORITY := 0);
    	PROGRAM instance0 WITH task0 : program0;
  	END_RESOURCE

END_CONFIGURATION

(* ---- IP_FIFO.ST ---- *)
TYPE
  oscat_IP_FIFO128_DATA  : ARRAY [1..128] OF BYTE;
  oscat_Mailbox  : ARRAY [1..16] OF BYTE;

  oscat_IP_FIFO_DATA :
  STRUCT
	X       : oscat_IP_FIFO128_DATA; (* IP_ID FIFO Speicher          *)
	Y       : oscat_IP_FIFO128_DATA; (* IP_ID Z�hler                 *)
	ID      : BYTE;                  (* h�chste vergabene id         *)
	MAX_ID  : BYTE;                  (* maximal Anmeldungen pro ID   *)
    INIT    : BOOL;                  (* Initialisierung durchgef�hrt *)
	EMPTY   : BOOL;                  (* FIFO leer                    *)
	FULL    : BOOL;                  (* FIFO voll                    *)
	TOP     : INT;                   (* maximale anzahl IN FIFO      *)
	NW      : INT;                   (* Schreibzeiger                *)
	NR      : INT;                   (* Lesezeiger                   *)
  END_STRUCT;
END_TYPE

TYPE

  oscat_NW_BUF_LONG  : ARRAY [0..4095] OF BYTE;

  oscat_NETWORK_BUFFER :
  STRUCT
    SIZE   : UINT;
    BUFFER : oscat_NW_BUF_LONG;
  END_STRUCT;

END_TYPE

FUNCTION _BYTE_TO_INT:INT
	VAR_INPUT
		IN :	BYTE;
	END_VAR

	_BYTE_TO_INT := USINT_TO_INT(BYTE_TO_USINT(IN));
END_FUNCTION

FUNCTION_BLOCK IP_FIFO_Block

  VAR_IN_OUT
    FIFO :	oscat_IP_FIFO_DATA;
    ID :	BYTE;
    STATE :	BYTE;
  END_VAR

  VAR
    tmp :	INT;
  END_VAR

  IF NOT FIFO.INIT THEN
    FIFO.INIT		:= TRUE;
    FIFO.NW		:= 1;
    FIFO.NR		:= 1;
    FIFO.EMPTY	:= TRUE;
    FIFO.FULL		:= FALSE;
    FIFO.TOP		:= 128;
    FIFO.MAX_ID	:= BYTE#1;
  END_IF;

  IF ID = BYTE#00 THEN
    IF FIFO.ID < INT_TO_BYTE(FIFO.TOP) THEN
      ID := USINT_TO_BYTE(BYTE_TO_USINT(FIFO.ID) + USINT#1);
      FIFO.ID := ID ;

    ELSIF STATE < BYTE#200 THEN
      STATE := BYTE#255;
    RETURN;
    END_IF;
  END_IF;

  IF STATE = BYTE#1 AND NOT FIFO.FULL THEN
    tmp := _BYTE_TO_INT(ID);
    IF FIFO.Y[tmp] < FIFO.MAX_ID THEN
      FIFO.Y[tmp] := USINT_TO_BYTE(BYTE_TO_USINT(FIFO.Y[tmp]) + USINT#1);
      tmp := FIFO.NW;
      FIFO.X[tmp] := ID;
      IF FIFO.NW = FIFO.TOP THEN FIFO.NW := 1; ELSE FIFO.NW := FIFO.NW + 1; END_IF;
      FIFO.FULL := FIFO.NW = FIFO.NR;
    FIFO.EMPTY := FALSE;
      STATE := BYTE#2;
    END_IF;
  END_IF;

  IF STATE = BYTE#2 AND NOT FIFO.EMPTY THEN
    tmp := FIFO.NR;
    IF ID = FIFO.X[tmp] THEN
      STATE := BYTE#3;
    END_IF;
  END_IF;

  IF STATE = BYTE#4 AND NOT FIFO.EMPTY THEN

    tmp := FIFO.NR;
    IF ID = FIFO.X[tmp] THEN
      tmp := _BYTE_TO_INT(ID);
      FIFO.Y[tmp] := USINT_TO_BYTE(BYTE_TO_USINT(FIFO.Y[tmp]) - USINT#1);

      IF FIFO.NR = FIFO.TOP THEN FIFO.NR := 1; ELSE FIFO.NR := FIFO.NR + 1; END_IF;
      FIFO.EMPTY := FIFO.NR = FIFO.NW;
    FIFO.FULL := FALSE;
    END_IF;
    STATE := BYTE#5;
  END_IF;

END_FUNCTION_BLOCK

PROGRAM program0
	VAR
		FIFO :	oscat_IP_FIFO_DATA;
    ID :	BYTE;
    STATE :	BYTE;

		func_block : IP_FIFO_Block;
	END_VAR
	func_block.FIFO := FIFO;
	func_block.ID := ID;
  func_block.STATE := STATE;

	func_block();
  FIFO  := func_block.FIFO;
	ID  := func_block.ID;
  STATE  := func_block.STATE;
END_PROGRAM

CONFIGURATION Config0
	RESOURCE ReS0 ON PLC
		TASK task0(INTERVAL := T#20ms,PRIORITY := 0);
		PROGRAM instance0 WITH task0 : program0;
	END_RESOURCE
END_CONFIGURATION

(* ---- IRTRANS_DECODE.ST ---- *)
FUNCTION_BLOCK CHR_TO_STRING_Block
	VAR_INPUT
		C :	BYTE;
	END_VAR

	VAR_OUTPUT
		CHR_TO_STRING :	STRING;
	END_VAR

	CHR_TO_STRING := BYTE_TO_STRING(C);

END_FUNCTION_BLOCK

TYPE

  oscat_NW_BUF_SHORT : ARRAY [0..1407] OF BYTE;
  oscat_NW_BUF_LONG  : ARRAY [0..4095] OF BYTE;

  oscat_NETWORK_BUFFER_SHORT :
  STRUCT
    SIZE   : UINT;
    BUFFER : oscat_NW_BUF_SHORT;
  END_STRUCT;

  oscat_NETWORK_BUFFER :
  STRUCT
    SIZE   : UINT;
    BUFFER : oscat_NW_BUF_LONG;
  END_STRUCT;

END_TYPE

TYPE
  oscat_IP_FIFO128_DATA  : ARRAY [1..128] OF BYTE;
  oscat_Mailbox  : ARRAY [1..16] OF BYTE;

  oscat_IP_FIFO_DATA :
  STRUCT
	X       : oscat_IP_FIFO128_DATA; (* IP_ID FIFO Speicher          *)
	Y       : oscat_IP_FIFO128_DATA; (* IP_ID Z�hler                 *)
	ID      : BYTE;                  (* h�chste vergabene id         *)
	MAX_ID  : BYTE;                  (* maximal Anmeldungen pro ID   *)
    INIT    : BOOL;                  (* Initialisierung durchgef�hrt *)
	EMPTY   : BOOL;                  (* FIFO leer                    *)
	FULL    : BOOL;                  (* FIFO voll                    *)
	TOP     : INT;                   (* maximale anzahl IN FIFO      *)
	NW      : INT;                   (* Schreibzeiger                *)
	NR      : INT;                   (* Lesezeiger                   *)
  END_STRUCT;

  oscat_IP_C:
  STRUCT
  	C_MODE:			BYTE;          		(*W Mode: TCP/UCP AKTIV/PASSIV                               *)
	C_PORT:         WORD;          		(*W Portnummer                                               *)
	C_IP:           DWORD;         		(*W IP-ADRESSe gepackt wwxxyyzz = www.xxx.yyy.zzz            *)
    C_STATE:        BYTE;          		(*R VerbindungsSTATUS ON/OFF + Flanke ON/OFF                 *)
	C_ENABLE:       BOOL;          		(*W Freigabe f�r Connect                                     *)
    R_OBSERVE:      BOOL;          		(*W Empfang ueberwachen                                      *)
    TIME_RESET:     BOOL;          		(*W Alle Timer ruecksetzen                                   *)
	ERROR:          DWORD;         		(*R vvwwxxyy (vv = CON_ERROR, ww = SEN_ERROR, xx = REC_ERROR *)
    FIFO:           oscat_IP_FIFO_DATA; (*I IP FIFO Struktur                                         *)
	MAILBOX:		oscat_Mailbox;		(*I Mailbox: Datenbereich f�r Bausteindatenaustausch         *)
  END_STRUCT;
END_TYPE

FUNCTION_BLOCK IRTRANS_DECODE_Block

	VAR_OUTPUT
		CMD :	BOOL;
		DEV :	STRING;
		KEY :	STRING;
		ERROR :	BOOL;
	END_VAR

	VAR_IN_OUT
		IP_C :	oscat_IP_C;
		R_BUF :	oscat_NETWORK_BUFFER;
	END_VAR

	VAR
		i :	INT;
		STOP :	INT;
		received_string :	STRING;
		CHAR :	STRING;
		CHR_TO_STRING :	CHR_TO_STRING_Block;
		z :	BYTE;
	END_VAR

	i := UINT_TO_INT(R_BUF.SIZE);
	IF i >= 5 AND (i <= 82) AND IP_C.MAILBOX[1] <> z THEN
		ERROR := TRUE;
		i := i - 1;

		IF R_BUF.BUFFER[i] <> BYTE#10 THEN RETURN; END_IF;
		i := i - 1;
		IF R_BUF.BUFFER[i] <> BYTE#13 THEN RETURN; END_IF;
		i := i - 1;

		STOP := 0;
		received_string := '';

		WHILE STOP <= i DO
			CHR_TO_STRING(C:=R_BUF.BUFFER[STOP]);
			CHAR := CHR_TO_STRING.CHR_TO_STRING;
			received_string := CONCAT(received_string,CHAR);
			STOP := STOP + INT#1;
		END_WHILE;

		STOP := FIND(received_string,',');
		IF STOP > 0 AND STOP - 1 < i THEN
			DEV := LEFT(received_string,STOP - 1);
			key := RIGHT(received_string,i - STOP + 1);
			IF LEN(DEV) = 0 OR LEN(key) = 0 THEN RETURN; END_IF;
			cmd := TRUE;
			ERROR := FALSE;
		END_IF;
	ELSE
		cmd := FALSE;
		ERROR := FALSE;
	END_IF;

	z := IP_C.MAILBOX[1];

END_FUNCTION_BLOCK

PROGRAM program0
	VAR
		IP_C :	oscat_IP_C;
		R_BUF :	oscat_NETWORK_BUFFER;
		CMD :	BOOL;
		DEV :	STRING;
		KEY :	STRING;
		ERROR :	BOOL;

		func_block : IRTRANS_DECODE_Block;
	END_VAR
	func_block.IP_C := IP_C;
	func_block.R_BUF := R_BUF;

	func_block();
	IP_C  := func_block.IP_C;
	R_BUF  := func_block.R_BUF;
	CMD  := func_block.CMD;
	DEV  := func_block.DEV;
	KEY  := func_block.KEY;
	ERROR  := func_block.ERROR;

END_PROGRAM

CONFIGURATION Config0

  	RESOURCE ReS0 ON PLC
    	TASK task0(INTERVAL := T#20ms,PRIORITY := 0);
    	PROGRAM instance0 WITH task0 : program0;
  	END_RESOURCE

END_CONFIGURATION

(* ---- IRTRANS_RCV_1.ST ---- *)
FUNCTION_BLOCK IRTRANS_RCV_1_Block

	VAR_INPUT
		CMD :	BOOL;
		DEV_CODE :	STRING;
		KEY_CODE :	STRING;
	END_VAR

	VAR_OUTPUT
		Q :	BOOL;
	END_VAR

	VAR_IN_OUT
		DEV :	STRING;
		KEY :	STRING;
	END_VAR

	Q := cmd AND EQ_STRING(dev_code,dev) AND EQ_STRING(key_code,key);

END_FUNCTION_BLOCK

PROGRAM program0
	VAR
		CMD :	BOOL;
		DEV :	STRING;
		KEY :	STRING;
		DEV_CODE :	STRING;
		KEY_CODE :	STRING;
		Q :	BOOL;

		func_block : IRTRANS_RCV_1_Block;
	END_VAR
	func_block.CMD := CMD;
	func_block.DEV := DEV;
	func_block.KEY := KEY;
	func_block.DEV_CODE := DEV_CODE;
	func_block.KEY_CODE := KEY_CODE;

	func_block();
	DEV  := func_block.DEV;
	KEY  := func_block.KEY;
	Q  := func_block.Q;

END_PROGRAM

CONFIGURATION Config0

  	RESOURCE ReS0 ON PLC
    	TASK task0(INTERVAL := T#20ms,PRIORITY := 0);
    	PROGRAM instance0 WITH task0 : program0;
  	END_RESOURCE

END_CONFIGURATION

(* ---- IRTRANS_RCV_4.ST ---- *)
FUNCTION_BLOCK IRTRANS_RCV_4_Block

	VAR_INPUT
		CMD :	BOOL;
	END_VAR

	VAR_IN_OUT
		DEV :	STRING;
		KEY :	STRING;
	END_VAR

	VAR_INPUT
		DEV_CODE :	STRING;
		KEY_CODE_0 :	STRING;
		KEY_CODE_1 :	STRING;
		KEY_CODE_2 :	STRING;
		KEY_CODE_3 :	STRING;
	END_VAR

	VAR_OUTPUT
		Q0 :	BOOL;
		Q1 :	BOOL;
		Q2 :	BOOL;
		Q3 :	BOOL;
	END_VAR

	VAR
		decode :	BOOL;
	END_VAR

	decode := cmd AND EQ_STRING(dev_code,dev);

	Q0 := EQ_STRING(key,key_code_0) AND decode;
	Q1 := EQ_STRING(key,key_code_1) AND decode;
	Q2 := EQ_STRING(key,key_code_2) AND decode;
	Q3 := EQ_STRING(key,key_code_3) AND decode;

END_FUNCTION_BLOCK

PROGRAM program0
	VAR
		CMD :	BOOL;
		DEV :	STRING;
		KEY :	STRING;
		DEV_CODE :	STRING;
		KEY_CODE_0 :	STRING;
		KEY_CODE_1 :	STRING;
		KEY_CODE_2 :	STRING;
		KEY_CODE_3 :	STRING;
		Q0 :	BOOL;
		Q1 :	BOOL;
		Q2 :	BOOL;
		Q3 :	BOOL;

		func_block : IRTRANS_RCV_4_Block;
	END_VAR
	func_block.CMD := CMD;
	func_block.DEV := DEV;
	func_block.KEY := KEY;
	func_block.DEV_CODE := DEV_CODE;
	func_block.KEY_CODE_0 := KEY_CODE_0;
	func_block.KEY_CODE_1 := KEY_CODE_1;
	func_block.KEY_CODE_2 := KEY_CODE_2;
	func_block.KEY_CODE_3 := KEY_CODE_3;

	func_block();
	DEV  := func_block.DEV;
	KEY  := func_block.KEY;
	Q0  := func_block.Q0;
	Q1  := func_block.Q1;
	Q2  := func_block.Q2;
	Q3  := func_block.Q3;

END_PROGRAM

CONFIGURATION Config0

  	RESOURCE ReS0 ON PLC
    	TASK task0(INTERVAL := T#20ms,PRIORITY := 0);
    	PROGRAM instance0 WITH task0 : program0;
  	END_RESOURCE

END_CONFIGURATION

(* ---- IRTRANS_RCV_8.ST ---- *)
FUNCTION_BLOCK IRTRANS_RCV_8_Block

	VAR_INPUT
		CMD :	BOOL;
	END_VAR

	VAR_IN_OUT
		DEV :	STRING;
		KEY :	STRING;
	END_VAR

	VAR_INPUT
		DEV_CODE :	STRING;
		KEY_CODE_0 :	STRING;
		KEY_CODE_1 :	STRING;
		KEY_CODE_2 :	STRING;
		KEY_CODE_3 :	STRING;
		KEY_CODE_4 :	STRING;
		KEY_CODE_5 :	STRING;
		KEY_CODE_6 :	STRING;
		KEY_CODE_7 :	STRING;
	END_VAR

	VAR_OUTPUT
		Q0 :	BOOL;
		Q1 :	BOOL;
		Q2 :	BOOL;
		Q3 :	BOOL;
		Q4 :	BOOL;
		Q5 :	BOOL;
		Q6 :	BOOL;
		Q7 :	BOOL;
	END_VAR

	VAR
		decode :	BOOL;
	END_VAR

	decode := cmd AND EQ_STRING(dev_code,dev);

	Q0 := EQ_STRING(key,key_code_0) AND decode;
	Q1 := EQ_STRING(key,key_code_1) AND decode;
	Q2 := EQ_STRING(key,key_code_2) AND decode;
	Q3 := EQ_STRING(key,key_code_3) AND decode;
	Q4 := EQ_STRING(key,key_code_4) AND decode;
	Q5 := EQ_STRING(key,key_code_5) AND decode;
	Q6 := EQ_STRING(key,key_code_6) AND decode;
	Q7 := EQ_STRING(key,key_code_7) AND decode;

END_FUNCTION_BLOCK

PROGRAM program0
	VAR
		CMD :	BOOL;
		DEV :	STRING;
		KEY :	STRING;
		DEV_CODE :	STRING;
		KEY_CODE_0 :	STRING;
		KEY_CODE_1 :	STRING;
		KEY_CODE_2 :	STRING;
		KEY_CODE_3 :	STRING;
		KEY_CODE_4 :	STRING;
		KEY_CODE_5 :	STRING;
		KEY_CODE_6 :	STRING;
		KEY_CODE_7 :	STRING;
		Q0 :	BOOL;
		Q1 :	BOOL;
		Q2 :	BOOL;
		Q3 :	BOOL;
		Q4 :	BOOL;
		Q5 :	BOOL;
		Q6 :	BOOL;
		Q7 :	BOOL;

		func_block : IRTRANS_RCV_8_Block;
	END_VAR
	func_block.CMD := CMD;
	func_block.DEV := DEV;
	func_block.KEY := KEY;
	func_block.DEV_CODE := DEV_CODE;
	func_block.KEY_CODE_0 := KEY_CODE_0;
	func_block.KEY_CODE_1 := KEY_CODE_1;
	func_block.KEY_CODE_2 := KEY_CODE_2;
	func_block.KEY_CODE_3 := KEY_CODE_3;
	func_block.KEY_CODE_4 := KEY_CODE_4;
	func_block.KEY_CODE_5 := KEY_CODE_5;
	func_block.KEY_CODE_6 := KEY_CODE_6;
	func_block.KEY_CODE_7 := KEY_CODE_7;

	func_block();
	DEV  := func_block.DEV;
	KEY  := func_block.KEY;
	Q0  := func_block.Q0;
	Q1  := func_block.Q1;
	Q2  := func_block.Q2;
	Q3  := func_block.Q3;
	Q4  := func_block.Q4;
	Q5  := func_block.Q5;
	Q6  := func_block.Q6;
	Q7  := func_block.Q7;

END_PROGRAM

CONFIGURATION Config0

  	RESOURCE ReS0 ON PLC
    	TASK task0(INTERVAL := T#20ms,PRIORITY := 0);
    	PROGRAM instance0 WITH task0 : program0;
  	END_RESOURCE

END_CONFIGURATION

(* ---- IRTRANS_SERVER.ST ---- *)
TYPE

  oscat_NW_BUF_SHORT : ARRAY [0..1407] OF BYTE;
  oscat_NW_BUF_LONG  : ARRAY [0..4095] OF BYTE;

  oscat_NETWORK_BUFFER_SHORT :
  STRUCT
    SIZE   : UINT;
    BUFFER : oscat_NW_BUF_SHORT;
  END_STRUCT;

  oscat_NETWORK_BUFFER :
  STRUCT
    SIZE   : UINT;
    BUFFER : oscat_NW_BUF_LONG;
  END_STRUCT;

END_TYPE

TYPE
  oscat_IP_FIFO128_DATA  : ARRAY [1..128] OF BYTE;
  oscat_Mailbox  : ARRAY [1..16] OF BYTE;

  oscat_IP_FIFO_DATA :
  STRUCT
	X       : oscat_IP_FIFO128_DATA; (* IP_ID FIFO Speicher          *)
	Y       : oscat_IP_FIFO128_DATA; (* IP_ID Z�hler                 *)
	ID      : BYTE;                  (* h�chste vergabene id         *)
	MAX_ID  : BYTE;                  (* maximal Anmeldungen pro ID   *)
    INIT    : BOOL;                  (* Initialisierung durchgef�hrt *)
	EMPTY   : BOOL;                  (* FIFO leer                    *)
	FULL    : BOOL;                  (* FIFO voll                    *)
	TOP     : INT;                   (* maximale anzahl IN FIFO      *)
	NW      : INT;                   (* Schreibzeiger                *)
	NR      : INT;                   (* Lesezeiger                   *)
  END_STRUCT;

  oscat_IP_C:
  STRUCT
  	C_MODE:			BYTE;          		(*W Mode: TCP/UCP AKTIV/PASSIV                               *)
	C_PORT:         WORD;          		(*W Portnummer                                               *)
	C_IP:           DWORD;         		(*W IP-ADRESSe gepackt wwxxyyzz = www.xxx.yyy.zzz            *)
    C_STATE:        BYTE;          		(*R VerbindungsSTATUS ON/OFF + Flanke ON/OFF                 *)
	C_ENABLE:       BOOL;          		(*W Freigabe f�r Connect                                     *)
    R_OBSERVE:      BOOL;          		(*W Empfang ueberwachen                                      *)
    TIME_RESET:     BOOL;          		(*W Alle Timer ruecksetzen                                   *)
	ERROR:          DWORD;         		(*R vvwwxxyy (vv = CON_ERROR, ww = SEN_ERROR, xx = REC_ERROR *)
    FIFO:           oscat_IP_FIFO_DATA; (*I IP FIFO Struktur                                         *)
	MAILBOX:		oscat_Mailbox;		(*I Mailbox: Datenbereich f�r Bausteindatenaustausch         *)
  END_STRUCT;
END_TYPE

FUNCTION_BLOCK IRTRANS_SERVER_Block

	VAR_INPUT
		UDP_TCP :	BOOL;
	END_VAR

	VAR_OUTPUT
		S_ENABLE :	BOOL;
		R_ENABLE :	BOOL;
		ERROR :	DWORD;
	END_VAR

	VAR_IN_OUT
		IP_C :	oscat_IP_C;
		S_BUF :	oscat_NETWORK_BUFFER;
		R_BUF :	oscat_NETWORK_BUFFER;
	END_VAR

	VAR
		t :	TON;
	END_VAR

	IF NOT IP_C.C_ENABLE THEN
		IP_C.C_PORT := WORD#0;
		IP_C.C_IP := DWORD#00;
		IP_C.C_MODE := SEL(UDP_TCP,BYTE#5,BYTE#4);
		IP_C.C_ENABLE := TRUE;
		IP_C.R_OBSERVE := FALSE;
		IP_C.TIME_RESET := TRUE;
		S_BUF.SIZE := UINT#0;
		R_BUF.SIZE := UINT#0;
	END_IF;

	R_ENABLE := IP_C.C_STATE > BYTE#127;
	S_ENABLE := R_ENABLE AND (IP_C.MAILBOX[1] > BYTE#0 OR IP_C.C_MODE <> BYTE#5);
	ERROR := IP_C.ERROR;

	t(IN:= IP_C.ERROR > DWORD#0, PT:=T#5s);
	IF t.Q THEN
		IP_C.TIME_RESET := TRUE;
	END_IF;

END_FUNCTION_BLOCK

PROGRAM program0
	VAR
		UDP_TCP :	BOOL;
		S_ENABLE :	BOOL;
		R_ENABLE :	BOOL;
		ERROR :	DWORD;
		IP_C :	oscat_IP_C;
		S_BUF :	oscat_NETWORK_BUFFER;
		R_BUF :	oscat_NETWORK_BUFFER;

		func_block : IRTRANS_SERVER_Block;
	END_VAR
	func_block.UDP_TCP := UDP_TCP;
	func_block.IP_C := IP_C;
	func_block.S_BUF := S_BUF;
	func_block.R_BUF := R_BUF;

	func_block();
	S_ENABLE  := func_block.S_ENABLE;
	R_ENABLE  := func_block.R_ENABLE;
	ERROR  := func_block.ERROR;
	IP_C  := func_block.IP_C;
	S_BUF  := func_block.S_BUF;
	R_BUF  := func_block.R_BUF;

END_PROGRAM

CONFIGURATION Config0

  	RESOURCE ReS0 ON PLC
    	TASK task0(INTERVAL := T#20ms,PRIORITY := 0);
    	PROGRAM instance0 WITH task0 : program0;
  	END_RESOURCE

END_CONFIGURATION

(* ---- LOG_VIEWPORT.ST ---- *)
TYPE
  oscat_STRING80             : STRING;
  oscat_STRING250             : STRING;
END_TYPE

TYPE
  PRINTF_DATA_250  	:  ARRAY [1..11]  OF oscat_STRING250;
  PRINTF_DATA_80 	:  ARRAY [1..11]  OF oscat_STRING80;
  LOG_250       	:  ARRAY [0..400] OF oscat_STRING250;
  LOG_80    		:  ARRAY [0..400] OF oscat_STRING80;
  LOG_OPTION		:  ARRAY [0..400] OF DWORD;

  us_LOG_CONTROL :
  STRUCT
    NEW_MSG              : oscat_STRING250;    (*W neue Nachricht f�r den Datenbuffer   *)
	NEW_MSG_OPTION 		 : DWORD;
    LEVEL                : BYTE;
	SIZE                 : INT;                (*R Anzahl der Strings im LOG_DATA       *)
	RESET                : BOOL;               (*W Nachrichtenbuffer l�schen            *)
    PRINTF               : PRINTF_DATA_250;    (*W Array PRINTF Parameter               *)
    MSG                  : LOG_250;            (*I Array Message                        *)
    MSG_OPTION           : LOG_OPTION;     	   (*I Array Message OPTion                 *)
	UPDATE_COUNT         : UINT;               (*R Updatez�hler                         *)
    IDX                  : INT;                (*R aktueller Nachrichten-Index          *)
	RING_MODE            : BOOL;               (*I Buffer�berlauf erkannt               *)
  END_STRUCT;

  us_LOG_CONTROL_80 :
  STRUCT
    NEW_MSG              : oscat_STRING80;     (*W neue Nachricht f�r den Datenbuffer   *)
	NEW_MSG_OPTION 		 : DWORD;
    LEVEL                : BYTE;
	SIZE                 : INT;                (*R Anzahl der Strings im LOG_DATA       *)
	RESET                : BOOL;               (*W Nachrichtenbuffer l�schen            *)
    PRINTF               : PRINTF_DATA_80;     (*W Array PRINTF Parameter               *)
    MSG                  : LOG_80;             (*I Array Message                        *)
    MSG_OPTION           : LOG_OPTION;     	   (*I Array Message OPTion                 *)
	UPDATE_COUNT         : UINT;               (*R Updatez�hler                         *)
    IDX                  : INT;                (*R aktueller Nachrichten-Index          *)
	RING_MODE            : BOOL;               (*I Buffer�berlauf erkannt               *)
  END_STRUCT;

  LINE_ARRAY 			: ARRAY [1..40] OF INT;

  us_LOG_VIEWPORT :
    STRUCT
     LINE_ARRAY          : LINE_ARRAY;
     COUNT               : INT;                (* Anzahl der sichtbaren Nachtrichten   *)
	 UPDATE_COUNT        : UINT;               (* Updatez�hler                         *)
     MOVE_TO_X           : INT;                (* Steuerung der Nachrichtenanzeige     *)
     UPDATE              : BOOL;               (* Daten wurden ge�ndert -> neuzeichnen *)
  END_STRUCT;

END_TYPE

FUNCTION_BLOCK LOG_VIEWPORT_Block

  VAR_IN_OUT
    LC :	us_LOG_CONTROL_80;
    LV :	us_LOG_VIEWPORT;
  END_VAR

  VAR
    POS :	INT;
    count :	INT;
    idx :	INT;
    base :	INT;
    update_POS :	BOOL;
  END_VAR

  IF LV.MOVE_TO_X <> 0 THEN
    CASE LV.MOVE_TO_X OF
    30000:
      POS := 1 ;
    30001:
      POS := LC.SIZE;
    30002:
      POS := POS + LV.COUNT;
    30003:
      POS := POS - LV.COUNT;
    ELSE
      POS := POS + LV.MOVE_TO_X;
    END_CASE;
    update_POS := TRUE;
    LV.MOVE_TO_X := 0;
  END_IF;

  IF (LV.UPDATE_COUNT <> LC.UPDATE_COUNT) OR update_POS THEN
    LV.UPDATE := TRUE;
    LV.UPDATE_COUNT := LC.UPDATE_COUNT;
    update_POS := FALSE;

    IF LC.RING_MODE THEN
      POS := LIMIT(1,POS,LC.SIZE - LV.COUNT + 1);
    ELSE
      IF LC.IDX > LV.COUNT THEN
        POS := LIMIT(1,POS,LC.IDX - LV.COUNT + 1);
      ELSE
        POS := 1;
      END_IF;
    END_IF;

    base := LC.IDX - POS - LV.COUNT + 1;
    IF LC.RING_MODE THEN
      FOR count:= 1 TO LV.COUNT DO
        idx := base + count;
        IF idx < 1 THEN
          idx := idx + LC.SIZE;
        END_IF;
      END_FOR;
    ELSE
      FOR count:= 1 TO LV.COUNT DO
        idx := base + count;
        IF idx < 1 THEN
          LV.LINE_ARRAY[count] := 0;
        ELSE
          LV.LINE_ARRAY[count] := idx;
        END_IF;
      END_FOR;
    END_IF;
  END_IF;

END_FUNCTION_BLOCK

PROGRAM program0
	VAR
		LC :	us_LOG_CONTROL_80;
    LV :	us_LOG_VIEWPORT;

		func_block : LOG_VIEWPORT_Block;
	END_VAR
	func_block.LC := LC;
	func_block.LV := LV;

	func_block();
  LC  := func_block.LC;
  LV  := func_block.LV;

END_PROGRAM

CONFIGURATION Config0

  	RESOURCE ReS0 ON PLC
    	TASK task0(INTERVAL := T#20ms,PRIORITY := 0);
    	PROGRAM instance0 WITH task0 : program0;
  	END_RESOURCE

END_CONFIGURATION

(* ---- MB_CLIENT.ST ---- *)
TYPE
  oscat_IP_FIFO128_DATA  : ARRAY [1..128] OF BYTE;
  oscat_Mailbox  : ARRAY [1..16] OF BYTE;

  oscat_IP_FIFO_DATA :
  STRUCT
	X       : oscat_IP_FIFO128_DATA; (* IP_ID FIFO Speicher          *)
	Y       : oscat_IP_FIFO128_DATA; (* IP_ID Z�hler                 *)
	ID      : BYTE;                  (* h�chste vergabene id         *)
	MAX_ID  : BYTE;                  (* maximal Anmeldungen pro ID   *)
    INIT    : BOOL;                  (* Initialisierung durchgef�hrt *)
	EMPTY   : BOOL;                  (* FIFO leer                    *)
	FULL    : BOOL;                  (* FIFO voll                    *)
	TOP     : INT;                   (* maximale anzahl IN FIFO      *)
	NW      : INT;                   (* Schreibzeiger                *)
	NR      : INT;                   (* Lesezeiger                   *)
  END_STRUCT;

  oscat_IP_C:
  STRUCT
  	C_MODE:			BYTE;          		(*W Mode: TCP/UCP AKTIV/PASSIV                               *)
	C_PORT:         WORD;          		(*W Portnummer                                               *)
	C_IP:           DWORD;         		(*W IP-ADRESSe gepackt wwxxyyzz = www.xxx.yyy.zzz            *)
    C_STATE:        BYTE;          		(*R VerbindungsSTATUS ON/OFF + Flanke ON/OFF                 *)
	C_ENABLE:       BOOL;          		(*W Freigabe f�r Connect                                     *)
    R_OBSERVE:      BOOL;          		(*W Empfang ueberwachen                                      *)
    TIME_RESET:     BOOL;          		(*W Alle Timer ruecksetzen                                   *)
	ERROR:          DWORD;         		(*R vvwwxxyy (vv = CON_ERROR, ww = SEN_ERROR, xx = REC_ERROR *)
    FIFO:           oscat_IP_FIFO_DATA; (*I IP FIFO Struktur                                         *)
	MAILBOX:		oscat_Mailbox;		(*I Mailbox: Datenbereich f�r Bausteindatenaustausch         *)
  END_STRUCT;
END_TYPE

TYPE
	oscat_aW0_255	: ARRAY [0..255] OF WORD;
	oscat_NW_BUF_SHORT : ARRAY [0..1407] OF BYTE;
	oscat_NW_BUF_LONG  : ARRAY [0..4095] OF BYTE;

	oscat_NETWORK_BUFFER_SHORT :
	STRUCT
		SIZE   : UINT;
		BUFFER : oscat_NW_BUF_SHORT;
	END_STRUCT;

	oscat_NETWORK_BUFFER :
	STRUCT
		SIZE   : UINT;
		BUFFER : oscat_NW_BUF_LONG;
	END_STRUCT;

END_TYPE

FUNCTION _BYTE_TO_INT:INT
	VAR_INPUT
		IN :	BYTE;
	END_VAR

	_BYTE_TO_INT := USINT_TO_INT(BYTE_TO_USINT(IN));
END_FUNCTION

FUNCTION_BLOCK IP_FIFO_Block

  VAR_IN_OUT
    FIFO :	oscat_IP_FIFO_DATA;
    ID :	BYTE;
    STATE :	BYTE;
  END_VAR

  VAR
    tmp :	INT;
  END_VAR

  IF NOT FIFO.INIT THEN
    FIFO.INIT		:= TRUE;
    FIFO.NW		:= 1;
    FIFO.NR		:= 1;
    FIFO.EMPTY	:= TRUE;
    FIFO.FULL		:= FALSE;
    FIFO.TOP		:= 128;
    FIFO.MAX_ID	:= BYTE#1;
  END_IF;

  IF ID = BYTE#00 THEN
    IF FIFO.ID < INT_TO_BYTE(FIFO.TOP) THEN
      ID := USINT_TO_BYTE(BYTE_TO_USINT(FIFO.ID) + USINT#1);
      FIFO.ID := ID ;

    ELSIF STATE < BYTE#200 THEN
      STATE := BYTE#255;
    RETURN;
    END_IF;
  END_IF;

  IF STATE = BYTE#1 AND NOT FIFO.FULL THEN
    tmp := _BYTE_TO_INT(ID);
    IF FIFO.Y[tmp] < FIFO.MAX_ID THEN
      FIFO.Y[tmp] := USINT_TO_BYTE(BYTE_TO_USINT(FIFO.Y[tmp]) + USINT#1);
      tmp := FIFO.NW;
      FIFO.X[tmp] := ID;
      IF FIFO.NW = FIFO.TOP THEN FIFO.NW := 1; ELSE FIFO.NW := FIFO.NW + 1; END_IF;
      FIFO.FULL := FIFO.NW = FIFO.NR;
    FIFO.EMPTY := FALSE;
      STATE := BYTE#2;
    END_IF;
  END_IF;

  IF STATE = BYTE#2 AND NOT FIFO.EMPTY THEN
    tmp := FIFO.NR;
    IF ID = FIFO.X[tmp] THEN
      STATE := BYTE#3;
    END_IF;
  END_IF;

  IF STATE = BYTE#4 AND NOT FIFO.EMPTY THEN

    tmp := FIFO.NR;
    IF ID = FIFO.X[tmp] THEN
      tmp := _BYTE_TO_INT(ID);
      FIFO.Y[tmp] := USINT_TO_BYTE(BYTE_TO_USINT(FIFO.Y[tmp]) - USINT#1);

      IF FIFO.NR = FIFO.TOP THEN FIFO.NR := 1; ELSE FIFO.NR := FIFO.NR + 1; END_IF;
      FIFO.EMPTY := FIFO.NR = FIFO.NW;
    FIFO.FULL := FALSE;
    END_IF;
    STATE := BYTE#5;
  END_IF;

END_FUNCTION_BLOCK

FUNCTION WORD_OF_BYTE:WORD
	VAR_INPUT
		B1 :	BYTE;
		B0 :	BYTE;
	END_VAR
	WORD_OF_BYTE := SHL(BYTE_TO_WORD(B1),8) OR BYTE_TO_WORD(B0);
END_FUNCTION

FUNCTION BIT_LOAD_W:WORD
	VAR_INPUT
		IN :	WORD;
		VAL :	BOOL;
		POS :	INT;
	END_VAR

	IF VAL THEN
		BIT_LOAD_W := IN OR SHL(WORD#1,POS);
	ELSE
		BIT_LOAD_W := IN AND (NOT SHL(WORD#1,POS));
	END_IF;
END_FUNCTION

FUNCTION_BLOCK MB_CLIENT_Block

	VAR_IN_OUT
		IP_C :	oscat_IP_C;
		S_BUF :	oscat_NETWORK_BUFFER_SHORT;
		R_BUF :	oscat_NETWORK_BUFFER_SHORT;
		DATA :	oscat_aW0_255;
	END_VAR

	VAR_INPUT
		DATA_SIZE :	INT;
		ENABLE :	BOOL;
		UDP :	BOOL;
		FC :	INT;
		UNIT_ID :	BYTE;
		R_ADDR :	INT;
		R_POINTS :	INT;
		R_DATA_ADR :	INT;
		R_DATA_BITPOS :	INT;
		W_ADDR :	INT;
		W_POINTS :	INT;
		W_DATA_ADR :	INT;
		W_DATA_BITPOS :	INT;
		DELAY :	TIME;
	END_VAR

	VAR_OUTPUT
		ERROR :	DWORD;
		BUSY :	BOOL;
	END_VAR

	VAR
		IP_STATE :	BYTE;
		IP_ID :	BYTE;
		IP_FIFO :	IP_FIFO_Block;
		mask :	DWORD;
		w_tmp :	WORD;
		idX1 :	INT;
		idX2 :	INT;
		STOP :	INT;
		i :	INT;
		BIT_POS :	INT;
		w_mask :	WORD;
		b_mask :	BYTE;
		count :	INT;
		STATE :	INT;
		Transaction_ID :	INT;
		Response :	INT;
		comp :	INT;
		TON_1 :	TON;
	END_VAR

	CASE STATE OF

	00:
		TON_1(IN:=ENABLE,PT:=DELAY);

		IF TON_1.Q OR DELAY = T#0s THEN
			TON_1(IN:=FALSE);
			STATE := 20;
			IP_STATE := BYTE#1;
		END_IF;

	20:
		IF IP_STATE = BYTE#3 THEN
			IP_C.C_PORT     := WORD#0;
			IP_C.C_IP       := DWORD#0;
			IP_C.C_MODE     := BOOL_TO_BYTE(UDP);
			IP_C.TIME_RESET := TRUE;
			IP_C.C_ENABLE   := TRUE;
			IP_C.R_OBSERVE  := TRUE;

			ERROR := DWORD#00;

			CASE FC OF

			1..2:
				IF R_POINTS <= 2000 THEN
					w_tmp := INT_TO_WORD(R_ADDR);
					S_BUF.BUFFER[08] := WORD_TO_BYTE(SHR(w_tmp,8));
					S_BUF.BUFFER[09] := WORD_TO_BYTE(w_tmp);
					w_tmp := INT_TO_WORD(R_POINTS);
					S_BUF.BUFFER[10] := WORD_TO_BYTE(SHR(w_tmp,8));
					S_BUF.BUFFER[11] := WORD_TO_BYTE(w_tmp);
					S_BUF.SIZE := UINT#12;
					Response :=	WORD_TO_INT(SHR(INT_TO_WORD(R_POINTS + 7),3));
					comp := 7;
				ELSE
					ERROR := DWORD#2;
				END_IF;
			3..4:
				IF R_POINTS <= 125 THEN
					w_tmp := INT_TO_WORD(R_ADDR);
					S_BUF.BUFFER[08] := WORD_TO_BYTE(SHR(w_tmp,8));
					S_BUF.BUFFER[09] := WORD_TO_BYTE(w_tmp);
					w_tmp := INT_TO_WORD(R_POINTS);
					S_BUF.BUFFER[10] := WORD_TO_BYTE(SHR(w_tmp,8));
					S_BUF.BUFFER[11] := WORD_TO_BYTE(w_tmp);

					S_BUF.SIZE := UINT#12;
					Response :=	WORD_TO_INT(SHL(w_tmp,1));
					comp := 7;
				ELSE
					ERROR := DWORD#2;
				END_IF;
			5:
				IF W_DATA_ADR <= DATA_SIZE THEN
					w_tmp := INT_TO_WORD(W_ADDR);
					S_BUF.BUFFER[08] := WORD_TO_BYTE(SHR(w_tmp,8));
					S_BUF.BUFFER[09] := WORD_TO_BYTE(w_tmp);
					S_BUF.BUFFER[10] := SEL((DATA[W_DATA_ADR] AND SHL(WORD#1,W_DATA_BITPOS))>WORD#00,BYTE#16#00,BYTE#16#FF);
					S_BUF.BUFFER[11] := BYTE#00;

					S_BUF.SIZE := UINT#12;
					Response :=	3;
					comp := 11;
				ELSE
					ERROR := DWORD#2;
				END_IF;
			6:
				IF W_DATA_ADR <= DATA_SIZE THEN
					w_tmp := INT_TO_WORD(W_ADDR);
					S_BUF.BUFFER[08] := WORD_TO_BYTE(SHR(w_tmp,8));
					S_BUF.BUFFER[09] := WORD_TO_BYTE(w_tmp);
					w_tmp := DATA[W_DATA_ADR];
					S_BUF.BUFFER[10] := WORD_TO_BYTE(SHR(w_tmp,8));
					S_BUF.BUFFER[11] := WORD_TO_BYTE(w_tmp);

					S_BUF.SIZE := UINT#12;
					Response :=	3;
					comp := 11;
				ELSE
					ERROR := DWORD#2;
				END_IF;
			15:
				IF (WORD_TO_INT(SHR(INT_TO_WORD(WORD_TO_INT(SHL(INT_TO_WORD(W_DATA_ADR),4)) + W_POINTS + W_DATA_BITPOS + 15),4)) <= DATA_SIZE) AND W_POINTS <= 1968 THEN
					w_tmp := INT_TO_WORD(W_ADDR);
					S_BUF.BUFFER[08] := WORD_TO_BYTE(SHR(w_tmp,8));
					S_BUF.BUFFER[09] := WORD_TO_BYTE(w_tmp);
					w_tmp := INT_TO_WORD(W_POINTS);
					S_BUF.BUFFER[10] := WORD_TO_BYTE(SHR(w_tmp,8));
					S_BUF.BUFFER[11] := WORD_TO_BYTE(w_tmp);
					S_BUF.BUFFER[12] := WORD_TO_BYTE(SHR(INT_TO_WORD(W_POINTS + 7),3));

					w_mask := SHL(WORD#1,W_DATA_BITPOS);
					BIT_POS := 0;
					w_tmp := WORD#00;
					idX1 := 12;
					idX2 := W_DATA_ADR;
					FOR i := 1 TO W_POINTS DO
						w_tmp :=BIT_LOAD_W(w_tmp,(DATA[idX2] AND w_mask)>WORD#0,BIT_POS);
						BIT_POS := BIT_POS + 1;
						IF BIT_POS > 7 OR i=W_POINTS THEN
							BIT_POS := 0;
							idX1 := idX1 + 1;
							S_BUF.BUFFER[idX1] := WORD_TO_BYTE(w_tmp);
							w_tmp := WORD#0;
						END_IF;
						w_mask := ROL(w_mask,1);
						IF w_mask = WORD#1 THEN
							idX2 := idX2 + 1;
						END_IF;
					END_FOR;
					S_BUF.SIZE := INT_TO_UINT(idX1+1);
					Response :=	3;
					comp := 11;
				ELSE
					ERROR := DWORD#2;
				END_IF;
			16:
				IF W_DATA_ADR + W_POINTS <= DATA_SIZE AND W_POINTS <= 123 THEN
					w_tmp := INT_TO_WORD(W_ADDR);
					S_BUF.BUFFER[08] := WORD_TO_BYTE(SHR(w_tmp,8));
					S_BUF.BUFFER[09] := WORD_TO_BYTE(w_tmp);
					w_tmp := INT_TO_WORD(W_POINTS);
					S_BUF.BUFFER[10] := WORD_TO_BYTE(SHR(w_tmp,8));
					S_BUF.BUFFER[11] := WORD_TO_BYTE(w_tmp);
					S_BUF.BUFFER[12] := SHL(S_BUF.BUFFER[11],1);

					idX1 := 11;
					count := W_DATA_ADR + W_POINTS - 1;
					FOR i := W_DATA_ADR TO count DO
						idX1 := idX1 + 2;
						idX2 := idX1 + 1;
						w_tmp := DATA[i];
						S_BUF.BUFFER[idX1] := WORD_TO_BYTE(SHR(w_tmp,8));
						S_BUF.BUFFER[idX2] := WORD_TO_BYTE(w_tmp);
					END_FOR;

					S_BUF.SIZE := INT_TO_UINT(idX2 + 1);
					Response := 3;
					comp := 11;
				ELSE
					ERROR := DWORD#2;
				END_IF;
			22:
				IF W_DATA_ADR + 2 <= DATA_SIZE THEN
					w_tmp := INT_TO_WORD(W_ADDR);
					S_BUF.BUFFER[08] := WORD_TO_BYTE(SHR(w_tmp,8));
					S_BUF.BUFFER[09] := WORD_TO_BYTE(w_tmp);
					idX1 := W_DATA_ADR;
					w_tmp := DATA[idX1];
					S_BUF.BUFFER[10] := WORD_TO_BYTE(SHR(w_tmp,8));
					S_BUF.BUFFER[11] := WORD_TO_BYTE(w_tmp);
					idX1 := idX1 +1;
					w_tmp := DATA[idX1];
					S_BUF.BUFFER[12] := WORD_TO_BYTE(SHR(w_tmp,8));
					S_BUF.BUFFER[13] := WORD_TO_BYTE(w_tmp);

					S_BUF.SIZE := UINT#14;
					Response :=	5;
					comp := 13;
				ELSE
					ERROR := DWORD#2;
				END_IF;
			23:
				IF W_DATA_ADR + W_POINTS <= DATA_SIZE AND W_POINTS <= 121 AND R_POINTS <= 125 THEN
					idX1 := 15;
					count := W_DATA_ADR + W_POINTS - 1;
					FOR i := W_DATA_ADR TO count DO
						idX1 := idX1 + 2;
						idX2 := idX1 + 1;
						w_tmp := DATA[i];
						S_BUF.BUFFER[idX1] := WORD_TO_BYTE(SHR(w_tmp,8));
						S_BUF.BUFFER[idX2] := WORD_TO_BYTE(w_tmp);
					END_FOR;

					w_tmp := INT_TO_WORD(W_ADDR);
					S_BUF.BUFFER[12] := WORD_TO_BYTE(SHR(w_tmp,8));
					S_BUF.BUFFER[13] := WORD_TO_BYTE(w_tmp);
					w_tmp := INT_TO_WORD(W_POINTS);
					S_BUF.BUFFER[14] := WORD_TO_BYTE(SHR(w_tmp,8));
					S_BUF.BUFFER[15] := WORD_TO_BYTE(w_tmp);
					S_BUF.BUFFER[16] := SHL(S_BUF.BUFFER[15],1);

					w_tmp := INT_TO_WORD(R_ADDR);
					S_BUF.BUFFER[08] := WORD_TO_BYTE(SHR(w_tmp,8));
					S_BUF.BUFFER[09] := WORD_TO_BYTE(w_tmp);
					w_tmp := INT_TO_WORD(R_POINTS);
					S_BUF.BUFFER[10] := WORD_TO_BYTE(SHR(w_tmp,8));
					S_BUF.BUFFER[11] := WORD_TO_BYTE(w_tmp);

					S_BUF.SIZE := INT_TO_UINT(idX2+1);
					Response :=	WORD_TO_INT(SHL(w_tmp,1));
					comp := 7;
				ELSE
					ERROR := DWORD#2;
				END_IF;

			ELSE
				ERROR := DWORD#00000001;
			END_CASE;

			IF ERROR = DWORD#00 THEN
				Transaction_ID := Transaction_ID + 1;
				w_tmp := UINT_TO_WORD(S_BUF.SIZE - UINT#6);
				S_BUF.BUFFER[0] := IP_ID;
				S_BUF.BUFFER[1] := INT_TO_BYTE(Transaction_ID);
				S_BUF.BUFFER[2] := BYTE#00;
				S_BUF.BUFFER[3] := BYTE#00;
				S_BUF.BUFFER[4] := WORD_TO_BYTE(SHR(w_tmp,8));
				S_BUF.BUFFER[5] := WORD_TO_BYTE(w_tmp);
				S_BUF.BUFFER[6] := UNIT_ID;
				S_BUF.BUFFER[7] := INT_TO_BYTE(FC);
				R_BUF.SIZE := UINT#0;
				STATE := 30;
			ELSE
				IP_STATE := BYTE#4;
				STATE := 00;
			END_IF;
		END_IF;

	30:
		IF IP_C.ERROR <> DWORD#00 THEN
			ERROR := IP_C.ERROR;
			IP_STATE := BYTE#4;
			STATE := 00;

		ELSIF S_BUF.SIZE = UINT#0 AND R_BUF.SIZE > UINT#0 THEN

			w_tmp := INT_TO_WORD(Response + 3);
			S_BUF.BUFFER[4] := WORD_TO_BYTE(SHR(w_tmp,8));
			S_BUF.BUFFER[5] := WORD_TO_BYTE(w_tmp);

			FOR i := 0 TO comp DO
				IF S_BUF.BUFFER[i] <> R_BUF.BUFFER[i] THEN EXIT; END_IF;
			END_FOR;

			IF R_BUF.SIZE >= UINT#9 AND R_BUF.BUFFER[7] > BYTE#128 THEN
				ERROR := BYTE_TO_DWORD(R_BUF.BUFFER[8]);
				IP_STATE := BYTE#4;
				STATE := 00;

			ELSIF R_BUF.SIZE = INT_TO_UINT(Response + 9) AND i > comp THEN
				mask := SHL(DWORD#1,FC);

				IF (mask AND DWORD#2#00000000_00000000_00000000_00000110) <> DWORD#0 THEN
					IF WORD_TO_INT(SHR(INT_TO_WORD(WORD_TO_INT(SHL(INT_TO_WORD(R_DATA_ADR),4)) + R_POINTS + R_DATA_BITPOS + 15),4)) <= DATA_SIZE THEN
						b_mask := BYTE#1;
						idX1 := 09;
						idX2 := R_DATA_ADR;
						BIT_POS := R_DATA_BITPOS;
						FOR i := 1 TO R_POINTS DO
							DATA[idX2]:=BIT_LOAD_W(DATA[idX2],(R_BUF.BUFFER[idX1] AND b_mask)>BYTE#0,BIT_POS);
							BIT_POS := BIT_POS + 1;
							IF BIT_POS > 15 THEN
								idX2 := idX2 + 1;
								BIT_POS := 0;
							END_IF;
							b_mask := ROL(b_mask,1);
							IF b_mask = BYTE#1 THEN
								idX1 := idX1 +1;
							END_IF;
						END_FOR;
					ELSE
						ERROR := DWORD#2;
					END_IF;

				ELSIF (mask AND DWORD#2#00000000_10000000_00000000_00011000) <> DWORD#0 THEN
					IF R_DATA_ADR + R_POINTS <= DATA_SIZE THEN
						STOP := R_DATA_ADR + R_POINTS -1 ;
						idX1 := 07;
						FOR i := R_DATA_ADR TO STOP DO
							idX1 := idX1 +2;
							idX2 := idX1 +1;
							DATA[i] := WORD_OF_BYTE(R_BUF.BUFFER[idX1],R_BUF.BUFFER[idX2]);
						END_FOR;
					ELSE
						ERROR := DWORD#2;
					END_IF;
				ELSIF (mask AND DWORD#2#11111111_00111110_01111111_10000001) > DWORD#0 THEN
					ERROR := DWORD#1;
				END_IF;
			ELSE
				ERROR := DWORD#3;
			END_IF;

			IP_STATE := BYTE#4;
			STATE := 00;
			R_BUF.SIZE := UINT#0;

		END_IF;

	END_CASE;

	IP_FIFO(FIFO:=IP_C.FIFO,STATE:=IP_STATE,ID:=IP_ID);
	IP_C.FIFO:=IP_FIFO.FIFO;
	IP_STATE := IP_FIFO.STATE;
	IP_ID:=IP_FIFO.ID;

	BUSY := IP_STATE = BYTE#3;

END_FUNCTION_BLOCK

PROGRAM program0
	VAR
		IP_C :	oscat_IP_C;
		S_BUF :	oscat_NETWORK_BUFFER_SHORT;
		R_BUF :	oscat_NETWORK_BUFFER_SHORT;
		DATA :	oscat_aW0_255;
		DATA_SIZE :	INT;
		ENABLE :	BOOL;
		UDP :	BOOL;
		FC :	INT;
		UNIT_ID :	BYTE;
		R_ADDR :	INT;
		R_POINTS :	INT;
		R_DATA_ADR :	INT;
		R_DATA_BITPOS :	INT;
		W_POINTS :	INT;
		W_DATA_ADR :	INT;
		W_DATA_BITPOS :	INT;
		DELAY :	TIME;
		ERROR :	DWORD;
		BUSY :	BOOL;

		func_block : MB_CLIENT_Block;
	END_VAR
	func_block.IP_C := IP_C;
	func_block.S_BUF := S_BUF;
	func_block.R_BUF := R_BUF;
	func_block.DATA := DATA;
	func_block.DATA_SIZE := DATA_SIZE;
	func_block.ENABLE := ENABLE;
	func_block.UDP := UDP;
	func_block.FC := FC;
	func_block.UNIT_ID := UNIT_ID;
	func_block.R_ADDR := R_ADDR;
	func_block.R_POINTS := R_POINTS;
	func_block.R_DATA_ADR := R_DATA_ADR;
	func_block.R_DATA_BITPOS := R_DATA_BITPOS;
	func_block.W_DATA_ADR := W_DATA_ADR;
	func_block.W_POINTS := W_POINTS;
	func_block.W_DATA_BITPOS := W_DATA_BITPOS;
	func_block.DELAY := DELAY;

	func_block();
  	IP_C  := func_block.IP_C;
	S_BUF  := func_block.S_BUF;
	R_BUF  := func_block.R_BUF;
	DATA  := func_block.DATA;
	ERROR  := func_block.ERROR;
	BUSY  := func_block.BUSY;

END_PROGRAM

CONFIGURATION Config0

	VAR_GLOBAL
		PLC_TICKS_PER_SEC :	INT;
		PLC_SYS_TICK_CNT :	DINT;
	END_VAR

  	RESOURCE ReS0 ON PLC
    	TASK task0(INTERVAL := T#20ms,PRIORITY := 0);
    	PROGRAM instance0 WITH task0 : program0;
  	END_RESOURCE

END_CONFIGURATION

(* ---- MB_SERVER.ST ---- *)
TYPE
	oscat_IP_FIFO128_DATA  : ARRAY [1..128] OF BYTE;
	oscat_Mailbox  : ARRAY [1..16] OF BYTE;

	oscat_NW_BUF_SHORT : ARRAY [0..1407] OF BYTE;
	oscat_NW_BUF_LONG  : ARRAY [0..4095] OF BYTE;

	oscat_IP_FIFO_DATA :
	STRUCT
		X       : oscat_IP_FIFO128_DATA; (* IP_ID FIFO Speicher          *)
		Y       : oscat_IP_FIFO128_DATA; (* IP_ID Z�hler                 *)
		ID      : BYTE;                  (* h�chste vergabene id         *)
		MAX_ID  : BYTE;                  (* maximal Anmeldungen pro ID   *)
		INIT    : BOOL;                  (* Initialisierung durchgef�hrt *)
		EMPTY   : BOOL;                  (* FIFO leer                    *)
		FULL    : BOOL;                  (* FIFO voll                    *)
		TOP     : INT;                   (* maximale anzahl IN FIFO      *)
		NW      : INT;                   (* Schreibzeiger                *)
		NR      : INT;                   (* Lesezeiger                   *)
	END_STRUCT;

	oscat_IP_C:
	STRUCT
		C_MODE:			BYTE;          		(*W Mode: TCP/UCP AKTIV/PASSIV                               *)
		C_PORT:         WORD;          		(*W Portnummer                                               *)
		C_IP:           DWORD;         		(*W IP-ADRESSe gepackt wwxxyyzz = www.xxx.yyy.zzz            *)
		C_STATE:        BYTE;          		(*R VerbindungsSTATUS ON/OFF + Flanke ON/OFF                 *)
		C_ENABLE:       BOOL;          		(*W Freigabe f�r Connect                                     *)
		R_OBSERVE:      BOOL;          		(*W Empfang ueberwachen                                      *)
		TIME_RESET:     BOOL;          		(*W Alle Timer ruecksetzen                                   *)
		ERROR:          DWORD;         		(*R vvwwxxyy (vv = CON_ERROR, ww = SEN_ERROR, xx = REC_ERROR *)
		FIFO:           oscat_IP_FIFO_DATA; (*I IP FIFO Struktur                                         *)
		MAILBOX:		oscat_Mailbox;		(*I Mailbox: Datenbereich f�r Bausteindatenaustausch         *)
	END_STRUCT;

	oscat_NETWORK_BUFFER :
	STRUCT
		SIZE   : UINT;
		BUFFER : oscat_NW_BUF_LONG;
	END_STRUCT;

	oscat_NETWORK_BUFFER_SHORT :
	STRUCT
	SIZE   : UINT;
	BUFFER : oscat_NW_BUF_SHORT;
	END_STRUCT;

	oscat_aW0_255	: ARRAY [0..255] OF WORD;
	oscat_VMAP_DATA :
	STRUCT
		FC       : DWORD;
		V_ADR    : INT;
		V_SIZE   : INT;
		P_ADR    : INT;
		TIME_OUT : TIME;
	END_STRUCT;

	oscat_MB_VMAP : ARRAY [1..10] OF oscat_VMAP_DATA;

	csv_parser_demo_col : ARRAY [1..4] OF REAL;
	csv_parser_demo     : ARRAY [1..2] OF csv_parser_demo_col;

END_TYPE

FUNCTION_BLOCK MB_VMAP_Block

	VAR_IN_OUT
		VMAP :	oscat_MB_VMAP;
	END_VAR

	VAR_INPUT
		FC :	INT;
		V_ADR :	INT;
		V_CNT :	INT;
		SIZE :	INT;
	END_VAR

	VAR_OUTPUT
		P_ADR :	INT;
		P_BIT :	INT;
		ERROR :	BYTE;
	END_VAR

	VAR
		i :	INT;
		VOPT :	DWORD;
		vadr :	INT;
		padr :	INT;
		mask :	DWORD;
		VSIZE :	INT;
		w_tmp :	WORD;
		i_tmp :	INT;
		init :	BOOL;
	END_VAR

	IF init = FALSE THEN
		init := TRUE;
		IF VMAP[1].FC = DWORD#0 THEN
			VMAP[1].FC := DWORD#16#FFFF_FFFF;
			VMAP[1].V_ADR := 0;
			VMAP[1].V_SIZE := 256;
			VMAP[1].P_ADR := 0;
		END_IF;
	END_IF;

	ERROR := BYTE#02;
	mask := SHL(DWORD#1,FC);

	IF (mask AND DWORD#2#00000000_01000000_00000000_01100000) <> DWORD#0 THEN
		V_CNT := 1;
	ELSIF V_CNT = 0 THEN
		RETURN;
	END_IF;

	FOR i := 1 TO 10 DO
		VOPT := VMAP[i].FC;
		IF (VOPT AND mask) <> DWORD#0 THEN
			vadr := VMAP[i].V_ADR;
			VSIZE := VMAP[i].V_SIZE;
			padr := VMAP[i].P_ADR;

			IF (mask AND DWORD#2#00000000_00000000_10000000_00100110) <> DWORD#0 THEN
				i_tmp := WORD_TO_INT(SHR(INT_TO_WORD(V_ADR + V_CNT -1),4))+1;
				IF i_tmp <= SIZE AND i_tmp <= VSIZE THEN
					w_tmp := INT_TO_WORD(V_ADR);
					P_ADR := WORD_TO_INT(SHR(w_tmp,4)) + padr;
					P_BIT := WORD_TO_INT(w_tmp AND WORD#16#000F);
					ERROR := BYTE#0;
					EXIT;
				END_IF;
			ELSIF (mask AND DWORD#2#00000000_11000001_00000000_01011000) <> DWORD#0 THEN
				IF V_ADR >= vadr AND V_ADR + V_CNT <= vadr + VSIZE THEN
					P_ADR := V_ADR - vadr + padr;
					IF P_ADR + V_CNT <= SIZE THEN
						ERROR := BYTE#0;
						EXIT;
					END_IF;
				END_IF;
			ELSE
				ERROR := BYTE#01;
				RETURN;
			END_IF;
		END_IF;
	END_FOR;

	IF ERROR = BYTE#0 THEN
		IF (mask AND DWORD#2#00000000_11000001_10000000_01100000) <> DWORD#0 THEN
			VMAP[i].TIME_OUT := T#1ms;
		END_IF;
	END_IF;

END_FUNCTION_BLOCK

FUNCTION _BYTE_TO_INT:INT
	VAR_INPUT
		IN :	BYTE;
	END_VAR

	_BYTE_TO_INT := USINT_TO_INT(BYTE_TO_USINT(IN));
END_FUNCTION

FUNCTION_BLOCK IP_FIFO_Block

  VAR_IN_OUT
    FIFO :	oscat_IP_FIFO_DATA;
    ID :	BYTE;
    STATE :	BYTE;
  END_VAR

  VAR
    tmp :	INT;
  END_VAR

  IF NOT FIFO.INIT THEN
    FIFO.INIT		:= TRUE;
    FIFO.NW		:= 1;
    FIFO.NR		:= 1;
    FIFO.EMPTY	:= TRUE;
    FIFO.FULL		:= FALSE;
    FIFO.TOP		:= 128;
    FIFO.MAX_ID	:= BYTE#1;
  END_IF;

  IF ID = BYTE#00 THEN
    IF FIFO.ID < INT_TO_BYTE(FIFO.TOP) THEN
      ID := USINT_TO_BYTE(BYTE_TO_USINT(FIFO.ID) + USINT#1);
      FIFO.ID := ID ;

    ELSIF STATE < BYTE#200 THEN
      STATE := BYTE#255;
    RETURN;
    END_IF;
  END_IF;

  IF STATE = BYTE#1 AND NOT FIFO.FULL THEN
    tmp := _BYTE_TO_INT(ID);
    IF FIFO.Y[tmp] < FIFO.MAX_ID THEN
      FIFO.Y[tmp] := USINT_TO_BYTE(BYTE_TO_USINT(FIFO.Y[tmp]) + USINT#1);
      tmp := FIFO.NW;
      FIFO.X[tmp] := ID;
      IF FIFO.NW = FIFO.TOP THEN FIFO.NW := 1; ELSE FIFO.NW := FIFO.NW + 1; END_IF;
      FIFO.FULL := FIFO.NW = FIFO.NR;
    FIFO.EMPTY := FALSE;
      STATE := BYTE#2;
    END_IF;
  END_IF;

  IF STATE = BYTE#2 AND NOT FIFO.EMPTY THEN
    tmp := FIFO.NR;
    IF ID = FIFO.X[tmp] THEN
      STATE := BYTE#3;
    END_IF;
  END_IF;

  IF STATE = BYTE#4 AND NOT FIFO.EMPTY THEN

    tmp := FIFO.NR;
    IF ID = FIFO.X[tmp] THEN
      tmp := _BYTE_TO_INT(ID);
      FIFO.Y[tmp] := USINT_TO_BYTE(BYTE_TO_USINT(FIFO.Y[tmp]) - USINT#1);

      IF FIFO.NR = FIFO.TOP THEN FIFO.NR := 1; ELSE FIFO.NR := FIFO.NR + 1; END_IF;
      FIFO.EMPTY := FIFO.NR = FIFO.NW;
    FIFO.FULL := FALSE;
    END_IF;
    STATE := BYTE#5;
  END_IF;

END_FUNCTION_BLOCK

FUNCTION _UDINT_TO_TIME:TIME

	VAR_INPUT
		IN :	UDINT;
	END_VAR

	_UDINT_TO_TIME := DINT_TO_TIME(UDINT_TO_DINT(IN));

END_FUNCTION

FUNCTION_BLOCK T_PLC_MS_block

	VAR_OUTPUT
		T_PLC_MS :	UDINT;
	END_VAR

	VAR
		PLC_TICKS_PER_SEC :	INT;
		PLC_SYS_TICK_CNT :	DINT;
	END_VAR

	VAR
		debug :	BOOL;(*Debug-Mode ON / OFF*)
		N :	INT;(*Debug-Faktor*)
		Offset :	UDINT;(*Debug-Offset*)
		temp :	DWORD := DWORD#1;(*Debug-Offset*)
		MODE :	BOOL;(*modus*)
		faktor :	UDINT;(*Systemtakt-Faktor*)
		init :	BOOL;
		v_plc_ticks_per_sec :	UDINT;
		base :	UDINT := UDINT#1000;
	END_VAR

	IF init = FALSE THEN
		v_plc_ticks_per_sec := INT_TO_UDINT(PLC_TICKS_PER_SEC);
		IF v_plc_ticks_per_sec = UDINT#1024 THEN
			faktor := UDINT#1;
			MODE := FALSE;
		ELSIF v_plc_ticks_per_sec > UDINT#0 THEN
			IF v_plc_ticks_per_sec <= base THEN
				faktor := base / v_plc_ticks_per_sec;
				MODE := FALSE;
			ELSE
				faktor := v_plc_ticks_per_sec / base;
				MODE := TRUE;
			END_IF;
		ELSE
			faktor := UDINT#1;
		END_IF;
		init := TRUE;
	END_IF;

	IF MODE THEN
		T_PLC_MS := DINT_TO_UDINT(PLC_SYS_TICK_CNT) / faktor;
	ELSE
		T_PLC_MS := DINT_TO_UDINT(PLC_SYS_TICK_CNT) * faktor;
	END_IF;

	IF debug THEN
		T_PLC_MS := (DWORD_TO_UDINT(SHL(UDINT_TO_DWORD(T_PLC_MS),N) OR SHL(temp,N)) - UDINT#1) + Offset;
	END_IF;

END_FUNCTION_BLOCK

FUNCTION WORD_OF_BYTE:WORD
	VAR_INPUT
		B1 :	BYTE;
		B0 :	BYTE;
	END_VAR
	WORD_OF_BYTE := SHL(BYTE_TO_WORD(B1),8) OR BYTE_TO_WORD(B0);
END_FUNCTION

FUNCTION BIT_LOAD_W:WORD
	VAR_INPUT
		IN :	WORD;
		VAL :	BOOL;
		POS :	INT;
	END_VAR

	IF VAL THEN
		BIT_LOAD_W := IN OR SHL(WORD#1,POS);
	ELSE
		BIT_LOAD_W := IN AND (NOT SHL(WORD#1,POS));
	END_IF;
END_FUNCTION

FUNCTION_BLOCK MB_SERVER_Block

	VAR_IN_OUT
		IP_C :	oscat_IP_C;
		S_BUF :	oscat_NETWORK_BUFFER_SHORT;
		R_BUF :	oscat_NETWORK_BUFFER_SHORT;
		VMAP :	oscat_MB_VMAP;
		DATA :	oscat_aW0_255;
	END_VAR

	VAR_INPUT
		DATA_SIZE :	INT;
		ENABLE :	BOOL;
		UDP :	BOOL;
	END_VAR

	VAR_OUTPUT
		ERROR :	DWORD;
	END_VAR

	VAR
		MB_VMAP :	MB_VMAP_Block;
		adR1  :	INT;
		adR2 :	INT;
		points :	INT;
		pointS2 :	INT;
		coils :	BYTE;
		mask :	BYTE;
		idX1 :	INT;
		idX2 :	INT;
		BIT_POS :	INT;
		count :	INT;
		fc :	INT;
		i :	INT;
		STATE :	INT;
		IP_STATE :	BYTE;
		IP_ID :	BYTE;
		IP_FIFO :	IP_FIFO_Block;
		w_tmp :	WORD;
		last_cycle :	TIME;
		TX :	TIME;
		T_PLC_MS :	T_PLC_MS_block;
		t :	TON;
		ip_ERROR :	BOOL;
	END_VAR

	T_PLC_MS();
	TX := UDINT_TO_TIME(T_PLC_MS.T_PLC_MS);

	FOR i := 1 TO 10 DO
		IF VMAP[i].TIME_OUT > T#0s THEN
			VMAP[i].TIME_OUT := VMAP[i].TIME_OUT + SUB_TIME(TX, last)_cycle;
		END_IF;
	END_FOR;
	last_cycle := TX;
	ip_ERROR := IP_C.ERROR > DWORD#0;

	CASE STATE OF

	00:
		IF ENABLE THEN
			STATE := 10;
			IP_STATE := BYTE#1;
		END_IF;

	10:
		IF IP_STATE = BYTE#3 THEN

			IP_C.C_PORT     := WORD#0;
			IP_C.C_IP       := DWORD#0;
			IP_C.C_MODE     := SEL(UDP,BYTE#4,BYTE#5);
			IP_C.TIME_RESET := TRUE;
			IP_C.C_ENABLE   := TRUE;
			IP_C.R_OBSERVE  := FALSE;
			STATE := 20;
		END_IF;

	20:	IF NOT ip_ERROR THEN
			IF S_BUF.SIZE = UINT#0 AND R_BUF.SIZE > UINT#6 THEN
				IF  R_BUF.SIZE = WORD_TO_UINT(WORD_OF_BYTE(R_BUF.BUFFER[4],R_BUF.BUFFER[5])) + UINT#6 THEN
					ERROR := DWORD#00;

					FOR i := 0 TO 13 DO
						S_BUF.BUFFER[i] := R_BUF.BUFFER[i];
					END_FOR;

					fc := _BYTE_TO_INT(R_BUF.BUFFER[7]);

					adR1  := WORD_TO_INT(WORD_OF_BYTE(R_BUF.BUFFER[8],R_BUF.BUFFER[9]));
					points := WORD_TO_INT(WORD_OF_BYTE(R_BUF.BUFFER[10],R_BUF.BUFFER[11]));

					MB_VMAP(VMAP:=VMAP,FC:=fc,V_ADR:=adR1 ,V_CNT:=points,SIZE:=DATA_SIZE);
					VMAP:=MB_VMAP.VMAP;
					adR1 :=MB_VMAP.P_ADR;
					BIT_POS:=MB_VMAP.P_BIT;
					ERROR:=BYTE_TO_DWORD(MB_VMAP.ERROR);

					IF ERROR = DWORD#0 THEN
						CASE fc OF

						1..2 :
							count := 9;
							coils := BYTE#0;
							mask := BYTE#1;
							FOR i := 1 TO points DO
								IF mask = BYTE#0 THEN
									mask := BYTE#1;
									S_BUF.BUFFER[count] := coils;
									coils := BYTE#0;
									count := count + 1;
								END_IF;
								IF (DATA[adR1 ] AND SHL(WORD#1,BIT_POS)) > WORD#0 THEN
									coils := coils OR mask;
								END_IF;

								BIT_POS := BIT_POS + 1;
								IF BIT_POS > 15 THEN
									adR1  := adR1  + 1;
									BIT_POS := 0;
								END_IF;

								mask := SHL(mask,1);
							END_FOR;
							S_BUF.BUFFER[Count] := coils;

							S_BUF.BUFFER[8] := INT_TO_BYTE(count - 8);
							S_BUF.SIZE := INT_TO_UINT(count + 1);

						3..4 :
							idX1 := 07;
							count := adR1  + points - 1;
							FOR i := adR1  TO count DO
								idX1 := idX1 + 2;
								idX2 := idX1 + 1;
								w_tmp := DATA[i];
								S_BUF.BUFFER[idX1] := WORD_TO_BYTE(SHR(w_tmp,8));
								S_BUF.BUFFER[idX2] := WORD_TO_BYTE(w_tmp);
							END_FOR;
							S_BUF.BUFFER[8] := SHL(INT_TO_BYTE(points),1);
							S_BUF.SIZE := INT_TO_UINT(idX2 + 1);
						5 :
							DATA[adR1 ]:=BIT_LOAD_W(DATA[adR1 ],R_BUF.BUFFER[10]>BYTE#0,BIT_POS);
							S_BUF.SIZE := UINT#12;
						6 :
							DATA[adR1 ] := WORD_OF_BYTE(R_BUF.BUFFER[10],R_BUF.BUFFER[11]);
							S_BUF.SIZE := UINT#12;
						15 :
							mask := BYTE#1;
							idX1 := 13;
							FOR i := 1 TO points DO
								DATA[adR1 ]:=BIT_LOAD_W(DATA[adR1 ],(R_BUF.BUFFER[idX1] AND mask)>BYTE#0,BIT_POS);
								BIT_POS := BIT_POS + 1;
								IF BIT_POS > 15 THEN
									adR1  := adR1  + 1;
									BIT_POS := 0;
								END_IF;
								mask := ROL(mask,1);
								IF mask = BYTE#1 THEN
									idX1 := idX1 +1;
								END_IF;
							END_FOR;
							S_BUF.SIZE := UINT#12;
						16 :
							idX1 := 11;
							count := adR1  + points -1;
							FOR i := adR1  TO Count DO
								idX1 := idX1 + 2;
								idX2 := idX1 + 1;
								Data[i] := WORD_OF_BYTE(R_BUF.BUFFER[idX1],R_BUF.BUFFER[idX2]);
							END_FOR;
							S_BUF.SIZE := UINT#12;
						22 :
							w_tmp := WORD_OF_BYTE(R_BUF.BUFFER[11],R_BUF.BUFFER[11]);
							DATA[adR1 ] := (DATA[adR1 ] AND w_tmp) OR (WORD_OF_BYTE(R_BUF.BUFFER[12],R_BUF.BUFFER[13]) AND (NOT w_tmp));
							S_BUF.SIZE := UINT#14;
						23 :
							adR2 := WORD_TO_INT(WORD_OF_BYTE(R_BUF.BUFFER[12],R_BUF.BUFFER[13]));
							pointS2 := WORD_TO_INT(WORD_OF_BYTE(R_BUF.BUFFER[14],R_BUF.BUFFER[15]));

							MB_VMAP(VMAP:=VMAP,FC:=16,V_ADR:=adR2,V_CNT:=pointS2,SIZE:=DATA_SIZE);
							VMAP:=MB_VMAP.VMAP;
							adR2:=MB_VMAP.P_ADR;
							ERROR:=BYTE_TO_DWORD(MB_VMAP.ERROR);

							IF ERROR = DWORD#0 THEN
								idX1 := 15;
								count := adR2 + pointS2 -1;
								FOR i := adR2 TO count DO
									idX1 := idX1 + 2;
									idX2 := idX1 + 1;
									Data[i] := WORD_OF_BYTE(R_BUF.BUFFER[idX1],R_BUF.BUFFER[idX2]);
								END_FOR;

								idX1 := 07;
								count := adR1  + points - 1;
								FOR i := adR1  TO count DO
									idX1 := idX1 + 2;
									idX2 := idX1 + 1;
									w_tmp := DATA[i];
									S_BUF.BUFFER[idX1] := WORD_TO_BYTE(SHR(w_tmp,8));
									S_BUF.BUFFER[idX2] := WORD_TO_BYTE(w_tmp);
								END_FOR;
								S_BUF.BUFFER[8] := SHL(INT_TO_BYTE(points),1);
								S_BUF.SIZE := INT_TO_UINT(idX2 + 1);

							END_IF;

						ELSE
							ERROR := DWORD#01;
						END_CASE;
					END_IF;
				END_IF;

				IF ERROR > DWORD#0 THEN
					S_BUF.BUFFER[7] := S_BUF.BUFFER[7] OR BYTE#2#1000_0000;
					S_BUF.BUFFER[8] := DWORD_TO_BYTE(ERROR);
					S_BUF.SIZE := UINT#9;
				END_IF;

				S_BUF.BUFFER[4] := BYTE#0;
				S_BUF.BUFFER[5] := UINT_TO_BYTE(S_BUF.SIZE - UINT#6);

			END_IF;
		ELSE
			ERROR := IP_C.ERROR;
		END_IF;

		t(IN:= ip_ERROR, PT:=T#5s);
		IF t.Q THEN
			IP_C.TIME_RESET := TRUE;
		END_IF;

		R_BUF.SIZE := UINT#0;

		IF ENABLE = FALSE THEN
			IP_STATE := BYTE#4;
			STATE := 00;
		END_IF;
	END_CASE;

	IP_FIFO(FIFO:=IP_C.FIFO,STATE:=IP_STATE,ID:=IP_ID);
	IP_C.FIFO:=IP_FIFO.FIFO;
	IP_STATE := IP_FIFO.STATE;
	IP_ID:=IP_FIFO.ID;

END_FUNCTION_BLOCK

PROGRAM program0
	VAR
		IP_C :	oscat_IP_C;
		S_BUF :	oscat_NETWORK_BUFFER_SHORT;
		R_BUF :	oscat_NETWORK_BUFFER_SHORT;
		VMAP :	oscat_MB_VMAP;
		DATA :	oscat_aW0_255;
		DATA_SIZE :	INT;
		ENABLE :	BOOL;
		UDP :	BOOL;
		ERROR :	DWORD;

		func_block : MB_SERVER_Block;
	END_VAR
	func_block.IP_C := IP_C;
	func_block.S_BUF := S_BUF;
	func_block.R_BUF := R_BUF;
	func_block.VMAP := VMAP;
	func_block.DATA := DATA;
	func_block.DATA_SIZE := DATA_SIZE;
	func_block.ENABLE := ENABLE;
	func_block.UDP := UDP;

	func_block();
  	IP_C  := func_block.IP_C;
	S_BUF  := func_block.S_BUF;
	R_BUF  := func_block.R_BUF;
	VMAP  := func_block.VMAP;
	DATA  := func_block.DATA;
	ERROR  := func_block.ERROR;

END_PROGRAM

CONFIGURATION Config0

	VAR_GLOBAL
		PLC_TICKS_PER_SEC :	INT;
		PLC_SYS_TICK_CNT :	DINT;
	END_VAR

  	RESOURCE ReS0 ON PLC
    	TASK task0(INTERVAL := T#20ms,PRIORITY := 0);
    	PROGRAM instance0 WITH task0 : program0;
  	END_RESOURCE

END_CONFIGURATION

(* ---- MB_VMAP.ST ---- *)
TYPE
  oscat_VMAP_DATA :
  STRUCT
	FC       : DWORD;
    V_ADR    : INT;
    V_SIZE   : INT;
    P_ADR    : INT;
	TIME_OUT : TIME;
  END_STRUCT;

  oscat_MB_VMAP : ARRAY [1..10] OF oscat_VMAP_DATA;

  csv_parser_demo_col : ARRAY [1..4] OF REAL;
  csv_parser_demo     : ARRAY [1..2] OF csv_parser_demo_col;

END_TYPE

FUNCTION_BLOCK MB_VMAP_Block

	VAR_IN_OUT
		VMAP :	oscat_MB_VMAP;
	END_VAR

	VAR_INPUT
		FC :	INT;
		V_ADR :	INT;
		V_CNT :	INT;
		SIZE :	INT;
	END_VAR

	VAR_OUTPUT
		P_ADR :	INT;
		P_BIT :	INT;
		ERROR :	BYTE;
	END_VAR

	VAR
		i :	INT;
		VOPT :	DWORD;
		vadr :	INT;
		padr :	INT;
		mask :	DWORD;
		VSIZE :	INT;
		w_tmp :	WORD;
		i_tmp :	INT;
		init :	BOOL;
	END_VAR

	IF init = FALSE THEN
		init := TRUE;
		IF VMAP[1].FC = DWORD#0 THEN
			VMAP[1].FC := DWORD#16#FFFF_FFFF;
			VMAP[1].V_ADR := 0;
			VMAP[1].V_SIZE := 256;
			VMAP[1].P_ADR := 0;
		END_IF;
	END_IF;

	ERROR := BYTE#02;
	mask := SHL(DWORD#1,FC);

	IF (mask AND DWORD#2#00000000_01000000_00000000_01100000) <> DWORD#0 THEN
		V_CNT := 1;
	ELSIF V_CNT = 0 THEN
		RETURN;
	END_IF;

	FOR i := 1 TO 10 DO
		VOPT := VMAP[i].FC;
		IF (VOPT AND mask) <> DWORD#0 THEN
			vadr := VMAP[i].V_ADR;
			VSIZE := VMAP[i].V_SIZE;
			padr := VMAP[i].P_ADR;

			IF (mask AND DWORD#2#00000000_00000000_10000000_00100110) <> DWORD#0 THEN
				i_tmp := WORD_TO_INT(SHR(INT_TO_WORD(V_ADR + V_CNT -1),4))+1;
				IF i_tmp <= SIZE AND i_tmp <= VSIZE THEN
					w_tmp := INT_TO_WORD(V_ADR);
					P_ADR := WORD_TO_INT(SHR(w_tmp,4)) + padr;
					P_BIT := WORD_TO_INT(w_tmp AND WORD#16#000F);
					ERROR := BYTE#0;
					EXIT;
				END_IF;
			ELSIF (mask AND DWORD#2#00000000_11000001_00000000_01011000) <> DWORD#0 THEN
				IF V_ADR >= vadr AND V_ADR + V_CNT <= vadr + VSIZE THEN
					P_ADR := V_ADR - vadr + padr;
					IF P_ADR + V_CNT <= SIZE THEN
						ERROR := BYTE#0;
						EXIT;
					END_IF;
				END_IF;
			ELSE
				ERROR := BYTE#01;
				RETURN;
			END_IF;
		END_IF;
	END_FOR;

	IF ERROR = BYTE#0 THEN
		IF (mask AND DWORD#2#00000000_11000001_10000000_01100000) <> DWORD#0 THEN
			VMAP[i].TIME_OUT := T#1ms;
		END_IF;
	END_IF;

END_FUNCTION_BLOCK

PROGRAM program0
	VAR
		VMAP :	oscat_MB_VMAP;
		FC :	INT;
		V_ADR :	INT;
		V_CNT :	INT;
		SIZE :	INT;
		P_ADR :	INT;
		P_BIT :	INT;
		ERROR :	BYTE;

		func_block : MB_VMAP_Block;
	END_VAR
	func_block.VMAP := VMAP;
	func_block.V_ADR := V_ADR;
	func_block.FC := FC;
	func_block.V_CNT := V_CNT;
	func_block.SIZE := SIZE;

	func_block();
  	VMAP  := func_block.VMAP;
	P_ADR  := func_block.P_ADR;
	P_BIT  := func_block.P_BIT;
	ERROR  := func_block.ERROR;
END_PROGRAM

CONFIGURATION Config0
	RESOURCE ReS0 ON PLC
		TASK task0(INTERVAL := T#20ms,PRIORITY := 0);
		PROGRAM instance0 WITH task0 : program0;
	END_RESOURCE
END_CONFIGURATION

(* ---- MOON_PHASE.ST ---- *)
FUNCTION TIME_TO_UDINT2:UDINT
	VAR_INPUT
		X :	TIME;
	END_VAR

	TIME_TO_UDINT2 := DINT_TO_UDINT(TIME_TO_DINT(X));
END_FUNCTION

FUNCTION_BLOCK MOON_PHASE_Block

	VAR_INPUT
		XDT :	UDINT;
		SCALE :	BYTE := BYTE#12;
		UPDATE :	TIME := T#1h;
	END_VAR

	VAR_OUTPUT
		PHASE :	BYTE;
	END_VAR

	VAR
		x :	UDINT;
		last_dt :	UDINT;
	END_VAR

	IF XDT - last_dt > TIME_TO_UDINT2(UPDATE) THEN
		x := (XDT - UDINT#603240) MOD UDINT#2551392;
		PHASE := UDINT_TO_BYTE(BYTE_TO_UDINT(SCALE) * x / UDINT#2551392) ;
		last_dt := XDT;
	END_IF;

END_FUNCTION_BLOCK

PROGRAM program0
	VAR
		XDT :	UDINT;
		SCALE :	BYTE := BYTE#12;
		UPDATE :	TIME := T#1h;
		PHASE :	BYTE;

		func_block : MOON_PHASE_Block;
	END_VAR
	func_block.XDT := XDT;
	func_block.SCALE := SCALE;
	func_block.UPDATE := UPDATE;

	func_block();
  	PHASE  := func_block.PHASE;
END_PROGRAM

CONFIGURATION Config0
	RESOURCE ReS0 ON PLC
		TASK task0(INTERVAL := T#20ms,PRIORITY := 0);
		PROGRAM instance0 WITH task0 : program0;
	END_RESOURCE
END_CONFIGURATION
